// TwinCAT 3 PLC project SxrVacPlc
// ProgramVersion: 3.1.4022.4
// libraries:
//   L2SI Vacuum Library, * (SLAC)
//   LCLS General, * (SLAC)
//   Tc2_Standard, * (Beckhoff Automation GmbH)
//   Tc2_System, * (Beckhoff Automation GmbH)
//   Tc2_Utilities, * (Beckhoff Automation GmbH)
//   Tc3_Module, * (Beckhoff Automation GmbH)
// project tree:
//   GVLs/ GVL_SXR_VAC.TcGVL, GVL_Variables.TcGVL
//   / PlcTask.TcTTO
//   POUs/ MAIN.TcPOU, PRG_DIAGNOSTIC.TcPOU, PRG_SXR_VAC.TcPOU
// real-time tasks:
//   TASK PlcTask: cycle T#10ms, priority 20, ADS port 350
//   TASK SimTask: cycle T#10ms, priority 21, ADS port 351
// I/O:
//   DEVICE =+-EK1200_00_00-CPU/EtherCAT1, AmsNetId 10.0.1.49.2.1
//     =+-EK1200_00_00 [EK1200-5000 EtherCAT Power supply (2A E-Bus)]
//       =+-ES3064_00_01 [EL3064 4Ch. Ana. Input 0-10V]
//       =+-ES1004_00_02 [EL1004 4Ch. Dig. Input 24V, 3ms]
//       =+-EL2794_00_03 [EL2794 4Ch. Dig. Output 24V AC/DC, 2A, short-circuit-proof]
//       =+-ES3064_00_04 [EL3064 4Ch. Ana. Input 0-10V]
//       =+-ES1004_00_05 [EL1004 4Ch. Dig. Input 24V, 3ms]
//       =+-EL2794_00_06 [EL2794 4Ch. Dig. Output 24V AC/DC, 2A, short-circuit-proof]
//       =+-EL9410_00_07 [EL9410 E-Bus Power Supplier  (Diagnostics)]
//       =+-ES3064_00_08 [EL3064 4Ch. Ana. Input 0-10V]
//       =+-ES1004_00_09 [EL1004 4Ch. Dig. Input 24V, 3ms]
//       =+-EL2794_00_10 [EL2794 4Ch. Dig. Output 24V AC/DC, 2A, short-circuit-proof]
//       =+-ES3064_00_11 [EL3064 4Ch. Ana. Input 0-10V]
//       =+-ES1004_00_12 [EL1004 4Ch. Dig. Input 24V, 3ms]
//       =+-EL2794_00_13 [EL2794 4Ch. Dig. Output 24V AC/DC, 2A, short-circuit-proof]
//       =+-EK1110_00_14 [EK1110 EtherCAT extension]
//     =+-EK1100_01_00 [EK1100 EtherCAT Coupler (2A E-Bus)]
//       =+-ES3068_01_01 [EL3068 8Ch. Ana. Input 0-10V]
//       =+-EL2798_01_02 [EL2798 8Ch. Dig. Output 24V AC/DC, 2A, potential-free]
//       =+-ES9187_01_03 [EL9187 Potential Connection, 8 x Ground]
//       =+-ES3068_01_04 [EL3068 8Ch. Ana. Input 0-10V]
//       =+-ES3068_01_05 [EL3068 8Ch. Ana. Input 0-10V]
//       =+-EL2798_01_06 [EL2798 8Ch. Dig. Output 24V AC/DC, 2A, potential-free]
//       =+-ES9187_01_07 [EL9187 Potential Connection, 8 x Ground]
//       =+-ES3068_01_08 [EL3068 8Ch. Ana. Input 0-10V]
//       =+-EL9410_01_09 [EL9410 E-Bus Power Supplier  (Diagnostics)]
//       =+-EL2202_01_10 [EL2022 2Ch. Dig. Output 24V, 2A]
//       =+-EL6695_01_11 [EL6695 EtherCAT Bridge terminal (Primary)]
//       =+-EL6695_01_12 [EL6695 EtherCAT Bridge terminal (Primary)]
//       =+-EL6695_01_13 [EL6695 EtherCAT Bridge terminal (Primary)]
//       =+-EL6695_01_14 [EL6695 EtherCAT Bridge terminal (Primary)]
//     =+-EK1100_02_00 [EK1100 EtherCAT Coupler (2A E-Bus)]
//       =+-EL3064_02_01 [EL3064 4Ch. Ana. Input 0-10V]
//       =+-EL9070_02_02 [EL9070 Shield terminal]
//       =+-ES1008_02_03 [EL1008 8Ch. Dig. Input 24V, 3ms]
//       =+-ES9184_02_04 [EL9184 Potential Connection, 8 x 24V, 8 x Ground]
//       =+-ES2008_02_05 [EL2008 8Ch. Dig. Output 24V, 0.5A]
//       =+-EL2798_02_06 [EL2798 8Ch. Dig. Output 24V AC/DC, 2A, potential-free]
//     =+-EK1100_03_00 [EK1100 EtherCAT Coupler (2A E-Bus)]
//       =+-ES1004_03_01 [EL1004 4Ch. Dig. Input 24V, 3ms]
//       =+-ES2004_03_02 [EL2004 4Ch. Dig. Output 24V, 0.5A]
//       =+-ES2004_03_03 [EL2004 4Ch. Dig. Output 24V, 0.5A]
//       =+-ES1004_03_04 [EL1008 8Ch. Dig. Input 24V, 3ms]
//       =+-EL3064_03_05 [EL3064 4Ch. Ana. Input 0-10V]
//       =+-EL9070_03_06 [EL9070 Shield terminal]
//       =+-ES1008_03_07 [EL1008 8Ch. Dig. Input 24V, 3ms]
//       =+-ES9184_03_08 [EL9184 Potential Connection, 8 x 24V, 8 x Ground]
//       =+-ES2008_03_09 [EL2008 8Ch. Dig. Output 24V, 0.5A]
//       =+-EL2798_03_10 [EL2798 8Ch. Dig. Output 24V AC/DC, 2A, potential-free]
//     =+-EP2338_04_00 [EP2338-0002 8 Ch. Dig. Input/Output 24V, 0,5A, M12]
//     =+-EP2338_05_00 [EP2338-0002 8 Ch. Dig. Input/Output 24V, 0,5A, M12]
//     =+-EK1100_05_01 [EK1100 EtherCAT Coupler (2A E-Bus)]
//       =+-ES1004_05_02 [EL1004 4Ch. Dig. Input 24V, 3ms]
//       =+-ES2202_05_03 [EL2202 2Ch. Dig. Output 24V, 0.5A]
//       =+-ES2202_05_04 [EL2202 2Ch. Dig. Output 24V, 0.5A]
//       =+-ES9505_05_05 [EL9505 Power supply terminal 5V]
//       =+-ES1124_05_06 [EL1124 4Ch. Dig. Input 5V, 10µs, Sensor Power]
//     =+-EP2338_06_00 [EP2338-0002 8 Ch. Dig. Input/Output 24V, 0,5A, M12]
//     =+-EP2338_07_00 [EP2338-0002 8 Ch. Dig. Input/Output 24V, 0,5A, M12]
//     =+-EP3174_07_01 [EP3174-0002 4Ch. Ana. Input +/-10V, 0-10V, 0/4-20mA configurable]
//     =+-EP2624_07_02 [EP2624-0002 4Ch. Relay Output, NO (125V AC / 30V DC)]
//     =+-EP2338_08_00 [EP2338-0002 8 Ch. Dig. Input/Output 24V, 0,5A, M12]
//     =+-EP3174_08_01 [EP3174-0002 4Ch. Ana. Input +/-10V, 0-10V, 0/4-20mA configurable]
//     =+-EP2624_08_02 [EP2624-0002 4Ch. Relay Output, NO (125V AC / 30V DC)]
//     =+-EP3174_09_00 [EP3174-0002 4Ch. Ana. Input +/-10V, 0-10V, 0/4-20mA configurable]
//     =+-EP2624_09_01 [EP2624-0002 4Ch. Relay Output, NO (125V AC / 30V DC)]
//     =+-EP2338_09_02 [EP2338-0002 8 Ch. Dig. Input/Output 24V, 0,5A, M12]
//     =+-EP2338_09_03 [EP2338-0002 8 Ch. Dig. Input/Output 24V, 0,5A, M12]
//     =+-EP3174_10_00 [EP3174-0002 4Ch. Ana. Input +/-10V, 0-10V, 0/4-20mA configurable]
//     =+-EP2624_10_01 [EP2624-0002 4Ch. Relay Output, NO (125V AC / 30V DC)]
//     =+-EP2338_10_02 [EP2338-0002 8 Ch. Dig. Input/Output 24V, 0,5A, M12]
//     =+-EP3174_11_00 [EP3174-0002 4Ch. Ana. Input +/-10V, 0-10V, 0/4-20mA configurable]
//     =+-EP2624_11_01 [EP2624-0002 4Ch. Relay Output, NO (125V AC / 30V DC)]
//     =+-EP2338_11_02 [EP2338-0002 8 Ch. Dig. Input/Output 24V, 0,5A, M12]
//     =+-EK1100_11_03 [EK1100 EtherCAT Coupler (2A E-Bus)]
//       =+-ES1004_11_04 [EL1004 4Ch. Dig. Input 24V, 3ms]
//       =+-ES2202_11_05 [EL2202 2Ch. Dig. Output 24V, 0.5A]
//       =+-ES2202_11_06 [EL2202 2Ch. Dig. Output 24V, 0.5A]
//       =+-ES9505_11_07 [EL9505 Power supply terminal 5V]
//       =+-ES1124_11_08 [EL1124 4Ch. Dig. Input 5V, 10µs, Sensor Power]
//     =+-EP3174_12_00 [EP3174-0002 4Ch. Ana. Input +/-10V, 0-10V, 0/4-20mA configurable]
//     =+-EP2624_12_01 [EP2624-0002 4Ch. Relay Output, NO (125V AC / 30V DC)]
//     =+-EP3174_13_00 [EP3174-0002 4Ch. Ana. Input +/-10V, 0-10V, 0/4-20mA configurable]
//     =+-EP2624_13_01 [EP2624-0002 4Ch. Relay Output, NO (125V AC / 30V DC)]
//     =+-EP2338_14_00 [EP2338-0002 8 Ch. Dig. Input/Output 24V, 0,5A, M12]
//     =+-EP3174_14_01 [EP3174-0002 4Ch. Ana. Input +/-10V, 0-10V, 0/4-20mA configurable]
//     =+-EP2624_14_02 [EP2624-0002 4Ch. Relay Output, NO (125V AC / 30V DC)]
//     =+-EK1100_15_00 [EK1100 EtherCAT Coupler (2A E-Bus)]
//       =+-ES3064_15_01 [EL3064 4Ch. Ana. Input 0-10V]
//       =+-ES1004_15_02 [EL1004 4Ch. Dig. Input 24V, 3ms]
//       =+-EL2794_15_03 [EL2794 4Ch. Dig. Output 24V AC/DC, 2A, short-circuit-proof]
//       =+-ES3064_15_04 [EL3064 4Ch. Ana. Input 0-10V]
//       =+-ES1004_15_05 [EL1004 4Ch. Dig. Input 24V, 3ms]
//       =+-EL2794_15_06 [EL2794 4Ch. Dig. Output 24V AC/DC, 2A, short-circuit-proof]
//   DEVICE SimDevice 2 (EtherCAT Simulation), AmsNetId 10.0.1.49.3.1
//     =+-ES3064_00_01 // EL3064-0000-0020
//     =+-ES1004_00_02 // EL1004-0000-0019
//     =+-EL2794_00_03 // EL2794-0000-0016
//     =+-ES3064_00_04 // EL3064-0000-0020
//     =+-ES1004_00_05 // EL1004-0000-0019
//     =+-EL2794_00_06 // EL2794-0000-0016
//     =+-EL9410_00_07 // EL9410-0000-0017
//     =+-ES3064_00_08 // EL3064-0000-0020
//     =+-ES1004_00_09 // EL1004-0000-0019
//     =+-EL2794_00_10 // EL2794-0000-0016
//     =+-ES3064_00_11 // EL3064-0000-0020
//     =+-ES1004_00_12 // EL1004-0000-0019
//     =+-EL2794_00_13 // EL2794-0000-0016
//     =+-EK1110_00_14 // EK1110-0000-0017
//     =+-EK1100_01_00 // EK1100-0000-0018
//     =+-ES3068_01_01 // EL3068-0000-0020
//     =+-EL2798_01_02 // EL2798-0000-0018
//     =+-ES3068_01_04 // EL3068-0000-0020
//     =+-ES3068_01_05 // EL3068-0000-0020
//     =+-EL2798_01_06 // EL2798-0000-0018
//     =+-ES3068_01_08 // EL3068-0000-0020
//     =+-EL9410_01_09 // EL9410-0000-0017
//     =+-EL2202_01_10 // EL2022-0000-0018
//     =+-EL6695_01_11 // EL6695-0000-0005
//     =+-EL6695_01_12 // EL6695-0000-0005
//     =+-EL6695_01_13 // EL6695-0000-0005
//     =+-EL6695_01_14 // EL6695-0000-0005
//     =+-EK1100_02_00 // EK1100-0000-0018
//     =+-EL3064_02_01 // EL3064-0000-0020
//     =+-ES1008_02_03 // EL1008-0000-0018
//     =+-ES2008_02_05 // EL2008-0000-0018
//     =+-EL2798_02_06 // EL2798-0000-0018
//     =+-EK1100_03_00 // EK1100-0000-0018
//     =+-ES1004_03_01 // EL1004-0000-0019
//     =+-ES2004_03_02 // EL2004-0000-0018
//     =+-ES2004_03_03 // EL2004-0000-0018
//     =+-ES1004_03_04 // EL1008-0000-0018
//     =+-EL3064_03_05 // EL3064-0000-0020
//     =+-ES1008_03_07 // EL1008-0000-0018
//     =+-ES2008_03_09 // EL2008-0000-0018
//     =+-EL2798_03_10 // EL2798-0000-0018
//     =+-EP2338_04_00 // EP2338-0002-0023
//     =+-EP2338_05_00 // EP2338-0002-0023
//     =+-EK1100_05_01 // EK1100-0000-0018
//     =+-ES1004_05_02 // EL1004-0000-0019
//     =+-ES2202_05_03 // EL2202-0000-0019
//     =+-ES2202_05_04 // EL2202-0000-0019
//     =+-ES9505_05_05 // EL9505-0000-0018
//     =+-ES1124_05_06 // EL1124-0000-0018
//     =+-EP2338_06_00 // EP2338-0002-0023
//     =+-EP2338_07_00 // EP2338-0002-0023
//     =+-EP3174_07_01 // EP3174-0002-0023
//     =+-EP2624_07_02 // EP2624-0002-0019
//     =+-EP2338_08_00 // EP2338-0002-0023
//     =+-EP3174_08_01 // EP3174-0002-0023
//     =+-EP2624_08_02 // EP2624-0002-0019
//     =+-EP3174_09_00 // EP3174-0002-0023
//     =+-EP2624_09_01 // EP2624-0002-0019
//     =+-EP2338_09_02 // EP2338-0002-0023
//     =+-EP2338_09_03 // EP2338-0002-0023
//     =+-EP3174_10_00 // EP3174-0002-0023
//     =+-EP2624_10_01 // EP2624-0002-0019
//     =+-EP2338_10_02 // EP2338-0002-0023
//     =+-EP3174_11_00 // EP3174-0002-0023
//     =+-EP2624_11_01 // EP2624-0002-0019
//     =+-EP2338_11_02 // EP2338-0002-0023
//     =+-EK1100_11_03 // EK1100-0000-0018
//     =+-ES1004_11_04 // EL1004-0000-0019
//     =+-ES2202_11_05 // EL2202-0000-0019
//     =+-ES2202_11_06 // EL2202-0000-0019
//     =+-ES9505_11_07 // EL9505-0000-0018
//     =+-ES1124_11_08 // EL1124-0000-0018
//     =+-EP3174_12_00 // EP3174-0002-0023
//     =+-EP2624_12_01 // EP2624-0002-0019
//     =+-EP3174_13_00 // EP3174-0002-0023
//     =+-EP2624_13_01 // EP2624-0002-0019
//     =+-EP2338_14_00 // EP2338-0002-0023
//     =+-EP3174_14_01 // EP3174-0002-0023
//     =+-EP2624_14_02 // EP2624-0002-0019
//     =+-EK1100_15_00 // EK1100-0000-0018
//     =+-ES3064_15_01 // EL3064-0000-0020
//     =+-ES1004_15_02 // EL1004-0000-0019
//     =+-EL2794_15_03 // EL2794-0000-0016
//     =+-ES3064_15_04 // EL3064-0000-0020
//     =+-ES1004_15_05 // EL1004-0000-0019
//     =+-EL2794_15_06 // EL2794-0000-0016
// variable links:
//   SxrVacPlc/SxrVacPlc Instance <-> =+-EK1200_00_00-CPU/EtherCAT1/=+-EK1100_01_00/=+-EL2798_01_02
//     PlcTask Outputs/GVL_SXR_VAC.fb_DMPS_GCC_1.q_xHV_DIS <-> Channel 1/GVL_SXR_VAC.fb_DMPS_GCC_1.q_xHV_DIS
//     PlcTask Outputs/GVL_SXR_VAC.fb_IM2K0_XTES_GCC_1.q_xHV_DIS <-> Channel 2/GVL_SXR_VAC.fb_IM2K0_XTES_GCC_1.q_xHV_DIS
//     PlcTask Outputs/GVL_SXR_VAC.fb_PCPM3B_GFS_1.q_xHV_DIS <-> Channel 5/GVL_SXR_VAC.fb_PCPM3B_GFS_1.q_xHV_DIS
//     PlcTask Outputs/GVL_SXR_VAC.fb_SL1K0_GCC_1.q_xHV_DIS <-> Channel 4/GVL_SXR_VAC.fb_SL1K0_GCC_1.q_xHV_DIS
//   SxrVacPlc/SxrVacPlc Instance <-> =+-EK1200_00_00-CPU/EtherCAT1/=+-EK1100_01_00/=+-EL2798_01_06
//     PlcTask Outputs/GVL_SXR_VAC.fb_MR1K1_BEND_GCC_1.q_xHV_DIS <-> Channel 5/GVL_SXR_VAC.fb_MR1K1_BEND_GCC_1.q_xHV_DIS
//     PlcTask Outputs/GVL_SXR_VAC.fb_PA1K0_GCC_1.q_xHV_DIS <-> Channel 4/GVL_SXR_VAC.fb_PA1K0_GCC_1.q_xHV_DIS
//     PlcTask Outputs/GVL_SXR_VAC.fb_TV2K0_GCC_1.q_xHV_DIS <-> Channel 1/GVL_SXR_VAC.fb_TV2K0_GCC_1.q_xHV_DIS
//     PlcTask Outputs/GVL_SXR_VAC.fb_TV2K0_GCC_2.q_xHV_DIS <-> Channel 2/GVL_SXR_VAC.fb_TV2K0_GCC_2.q_xHV_DIS
//   SxrVacPlc/SxrVacPlc Instance <-> =+-EK1200_00_00-CPU/EtherCAT1/=+-EK1100_01_00/=+-ES3068_01_01
//     PlcTask Inputs/GVL_SXR_VAC.fb_DMPS_GCC_1.i_iPRESS_R <-> AI Standard Channel 1/GVL_SXR_VAC.fb_DMPS_GCC_1.i_iPRESS_R
//     PlcTask Inputs/GVL_SXR_VAC.fb_DMPS_GPI_1.i_iPRESS_R <-> AI Standard Channel 5/GVL_SXR_VAC.fb_DMPS_GPI_1.i_iPRESS_R
//     PlcTask Inputs/GVL_SXR_VAC.fb_IM2K0_XTES_GCC_1.i_iPRESS_R <-> AI Standard Channel 3/GVL_SXR_VAC.fb_IM2K0_XTES_GCC_1.i_iPRESS_R
//     PlcTask Inputs/GVL_SXR_VAC.fb_IM2K0_XTES_GPI_1.i_iPRESS_R <-> AI Standard Channel 6/GVL_SXR_VAC.fb_IM2K0_XTES_GPI_1.i_iPRESS_R
//   SxrVacPlc/SxrVacPlc Instance <-> =+-EK1200_00_00-CPU/EtherCAT1/=+-EK1100_01_00/=+-ES3068_01_04
//     PlcTask Inputs/GVL_SXR_VAC.fb_PCPM3B_GFS_1.i_iPRESS_R <-> AI Standard Channel 3/GVL_SXR_VAC.fb_PCPM3B_GFS_1.i_iPRESS_R
//     PlcTask Inputs/GVL_SXR_VAC.fb_SL1K0_GCC_1.i_iPRESS_R <-> AI Standard Channel 1/GVL_SXR_VAC.fb_SL1K0_GCC_1.i_iPRESS_R
//     PlcTask Inputs/GVL_SXR_VAC.fb_SL1K0_GPI_1.i_iPRESS_R <-> AI Standard Channel 5/GVL_SXR_VAC.fb_SL1K0_GPI_1.i_iPRESS_R
//   SxrVacPlc/SxrVacPlc Instance <-> =+-EK1200_00_00-CPU/EtherCAT1/=+-EK1100_01_00/=+-ES3068_01_05
//     PlcTask Inputs/GVL_SXR_VAC.fb_TV2K0_GCC_1.i_iPRESS_R <-> AI Standard Channel 1/GVL_SXR_VAC.fb_TV2K0_GCC_1.i_iPRESS_R
//     PlcTask Inputs/GVL_SXR_VAC.fb_TV2K0_GCC_2.i_iPRESS_R <-> AI Standard Channel 3/GVL_SXR_VAC.fb_TV2K0_GCC_2.i_iPRESS_R
//     PlcTask Inputs/GVL_SXR_VAC.fb_TV2K0_GPI_1.i_iPRESS_R <-> AI Standard Channel 5/GVL_SXR_VAC.fb_TV2K0_GPI_1.i_iPRESS_R
//     PlcTask Inputs/GVL_SXR_VAC.fb_TV2K0_GPI_2.i_iPRESS_R <-> AI Standard Channel 6/GVL_SXR_VAC.fb_TV2K0_GPI_2.i_iPRESS_R
//   SxrVacPlc/SxrVacPlc Instance <-> =+-EK1200_00_00-CPU/EtherCAT1/=+-EK1100_01_00/=+-ES3068_01_08
//     PlcTask Inputs/GVL_SXR_VAC.fb_MR1K1_BEND_GCC_1.i_iPRESS_R <-> AI Standard Channel 3/GVL_SXR_VAC.fb_MR1K1_BEND_GCC_1.i_iPRESS_R
//     PlcTask Inputs/GVL_SXR_VAC.fb_MR1K1_BEND_GPI_1.i_iPRESS_R <-> AI Standard Channel 6/GVL_SXR_VAC.fb_MR1K1_BEND_GPI_1.i_iPRESS_R
//     PlcTask Inputs/GVL_SXR_VAC.fb_PA1K0_GCC_1.i_iPRESS_R <-> AI Standard Channel 1/GVL_SXR_VAC.fb_PA1K0_GCC_1.i_iPRESS_R
//     PlcTask Inputs/GVL_SXR_VAC.fb_PA1K0_GPI_1.i_iPRESS_R <-> AI Standard Channel 5/GVL_SXR_VAC.fb_PA1K0_GPI_1.i_iPRESS_R
//   SxrVacPlc/SxrVacPlc Instance <-> =+-EK1200_00_00-CPU/EtherCAT1/=+-EK1100_03_00/=+-ES1004_03_01
//     PlcTask Inputs/GVL_SXR_VAC.fb_EM1K0_GMD_VGC_1.i_xClsLS <-> Channel 4/GVL_SXR_VAC.fb_EM1K0_GMD_VGC_1.i_xClsLS
//     PlcTask Inputs/GVL_SXR_VAC.fb_EM1K0_GMD_VGC_1.i_xOpnLS <-> Channel 3/GVL_SXR_VAC.fb_EM1K0_GMD_VGC_1.i_xOpnLS
//     PlcTask Inputs/GVL_SXR_VAC.fb_RTDSK0_VGC_1.i_xClsLS <-> Channel 2/GVL_SXR_VAC.fb_RTDSK0_VGC_1.i_xClsLS
//     PlcTask Inputs/GVL_SXR_VAC.fb_RTDSK0_VGC_1.i_xOpnLS <-> Channel 1/GVL_SXR_VAC.fb_RTDSK0_VGC_1.i_xOpnLS
//   SxrVacPlc/SxrVacPlc Instance <-> =+-EK1200_00_00-CPU/EtherCAT1/=+-EK1100_03_00/=+-ES1004_03_04
//     PlcTask Inputs/GVL_SXR_VAC.fb_AT1K0_GAS_VGC_1.i_xClsLS <-> Channel 2/GVL_SXR_VAC.fb_AT1K0_GAS_VGC_1.i_xClsLS
//     PlcTask Inputs/GVL_SXR_VAC.fb_AT1K0_GAS_VGC_1.i_xOpnLS <-> Channel 1/GVL_SXR_VAC.fb_AT1K0_GAS_VGC_1.i_xOpnLS
//   SxrVacPlc/SxrVacPlc Instance <-> =+-EK1200_00_00-CPU/EtherCAT1/=+-EK1100_03_00/=+-ES2004_03_02
//     PlcTask Outputs/GVL_SXR_VAC.fb_EM1K0_GMD_VGC_1.q_xOPN_DO <-> Channel 3/GVL_SXR_VAC.fb_EM1K0_GMD_VGC_1.q_xOPN_DO
//     PlcTask Outputs/GVL_SXR_VAC.fb_RTDSK0_VGC_1.q_xOPN_DO <-> Channel 1/GVL_SXR_VAC.fb_RTDSK0_VGC_1.q_xOPN_DO
//   SxrVacPlc/SxrVacPlc Instance <-> =+-EK1200_00_00-CPU/EtherCAT1/=+-EK1100_03_00/=+-ES2004_03_03
//     PlcTask Outputs/GVL_SXR_VAC.fb_AT1K0_GAS_VGC_1.q_xOPN_DO <-> Channel 1/GVL_SXR_VAC.fb_AT1K0_GAS_VGC_1.q_xOPN_DO
//   SxrVacPlc/SxrVacPlc Instance <-> =+-EK1200_00_00-CPU/EtherCAT1/=+-EK1100_15_00/=+-EL2794_15_03
//     PlcTask Outputs/GVL_SXR_VAC.fb_MR1K4_SOMS_PIP_1.q_xHVEna_DO <-> Channel 1/GVL_SXR_VAC.fb_MR1K4_SOMS_PIP_1.q_xHVEna_DO
//     PlcTask Outputs/GVL_SXR_VAC.fb_ST1K4_TEST_PIP_1.q_xHVEna_DO <-> Channel 2/GVL_SXR_VAC.fb_ST1K4_TEST_PIP_1.q_xHVEna_DO
//     PlcTask Outputs/GVL_SXR_VAC.fb_ST2K4_BCS_PIP_1.q_xHVEna_DO <-> Channel 3/GVL_SXR_VAC.fb_ST2K4_BCS_PIP_1.q_xHVEna_DO
//     PlcTask Outputs/GVL_SXR_VAC.fb_ST3K4_PPS_PIP_1.q_xHVEna_DO <-> Channel 4/GVL_SXR_VAC.fb_ST3K4_PPS_PIP_1.q_xHVEna_DO
//   SxrVacPlc/SxrVacPlc Instance <-> =+-EK1200_00_00-CPU/EtherCAT1/=+-EK1100_15_00/=+-EL2794_15_06
//     PlcTask Outputs/GVL_SXR_VAC.fb_PC4K4_XTES_PIP_1.q_xHVEna_DO <-> Channel 1/GVL_SXR_VAC.fb_PC4K4_XTES_PIP_1.q_xHVEna_DO
//   SxrVacPlc/SxrVacPlc Instance <-> =+-EK1200_00_00-CPU/EtherCAT1/=+-EK1100_15_00/=+-ES1004_15_02
//     PlcTask Inputs/GVL_SXR_VAC.fb_MR1K4_SOMS_PIP_1.i_xSP_DI <-> Channel 1/GVL_SXR_VAC.fb_MR1K4_SOMS_PIP_1.i_xSP_DI
//     PlcTask Inputs/GVL_SXR_VAC.fb_ST1K4_TEST_PIP_1.i_xSP_DI <-> Channel 2/GVL_SXR_VAC.fb_ST1K4_TEST_PIP_1.i_xSP_DI
//     PlcTask Inputs/GVL_SXR_VAC.fb_ST2K4_BCS_PIP_1.i_xSP_DI <-> Channel 3/GVL_SXR_VAC.fb_ST2K4_BCS_PIP_1.i_xSP_DI
//     PlcTask Inputs/GVL_SXR_VAC.fb_ST3K4_PPS_PIP_1.i_xSP_DI <-> Channel 4/GVL_SXR_VAC.fb_ST3K4_PPS_PIP_1.i_xSP_DI
//   SxrVacPlc/SxrVacPlc Instance <-> =+-EK1200_00_00-CPU/EtherCAT1/=+-EK1100_15_00/=+-ES1004_15_05
//     PlcTask Inputs/GVL_SXR_VAC.fb_PC4K4_XTES_PIP_1.i_xSP_DI <-> Channel 1/GVL_SXR_VAC.fb_PC4K4_XTES_PIP_1.i_xSP_DI
//   SxrVacPlc/SxrVacPlc Instance <-> =+-EK1200_00_00-CPU/EtherCAT1/=+-EK1100_15_00/=+-ES3064_15_01
//     PlcTask Inputs/GVL_SXR_VAC.fb_MR1K4_SOMS_PIP_1.i_iPRESS <-> AI Standard Channel 1/GVL_SXR_VAC.fb_MR1K4_SOMS_PIP_1.i_iPRESS
//     PlcTask Inputs/GVL_SXR_VAC.fb_ST1K4_TEST_PIP_1.i_iPRESS <-> AI Standard Channel 2/GVL_SXR_VAC.fb_ST1K4_TEST_PIP_1.i_iPRESS
//     PlcTask Inputs/GVL_SXR_VAC.fb_ST2K4_BCS_PIP_1.i_iPRESS <-> AI Standard Channel 3/GVL_SXR_VAC.fb_ST2K4_BCS_PIP_1.i_iPRESS
//     PlcTask Inputs/GVL_SXR_VAC.fb_ST3K4_PPS_PIP_1.i_iPRESS <-> AI Standard Channel 4/GVL_SXR_VAC.fb_ST3K4_PPS_PIP_1.i_iPRESS
//   SxrVacPlc/SxrVacPlc Instance <-> =+-EK1200_00_00-CPU/EtherCAT1/=+-EK1100_15_00/=+-ES3064_15_04
//     PlcTask Inputs/GVL_SXR_VAC.fb_PC4K4_XTES_PIP_1.i_iPRESS <-> AI Standard Channel 1/GVL_SXR_VAC.fb_PC4K4_XTES_PIP_1.i_iPRESS
//   SxrVacPlc/SxrVacPlc Instance <-> =+-EK1200_00_00-CPU/EtherCAT1/=+-EK1200_00_00/=+-EL2794_00_03
//     PlcTask Outputs/GVL_SXR_VAC.fb_RTDSK0_PIP_{1..4}.q_xHVEna_DO <-> Channel {1..4}/GVL_SXR_VAC.fb_RTDSK0_PIP_{1..4}.q_xHVEna_DO  (4 links)
//   SxrVacPlc/SxrVacPlc Instance <-> =+-EK1200_00_00-CPU/EtherCAT1/=+-EK1200_00_00/=+-EL2794_00_06
//     PlcTask Outputs/GVL_SXR_VAC.fb_PCPM3B_PIP_1.q_xHVEna_DO <-> Channel 2/GVL_SXR_VAC.fb_PCPM3B_PIP_1.q_xHVEna_DO
//     PlcTask Outputs/GVL_SXR_VAC.fb_RTDSK0_PIP_5.q_xHVEna_DO <-> Channel 1/GVL_SXR_VAC.fb_RTDSK0_PIP_5.q_xHVEna_DO
//   SxrVacPlc/SxrVacPlc Instance <-> =+-EK1200_00_00-CPU/EtherCAT1/=+-EK1200_00_00/=+-EL2794_00_10
//     PlcTask Outputs/GVL_SXR_VAC.fb_MR1K1_BEND_PIP_1.q_xHVEna_DO <-> Channel 3/GVL_SXR_VAC.fb_MR1K1_BEND_PIP_1.q_xHVEna_DO
//     PlcTask Outputs/GVL_SXR_VAC.fb_MR1K3_TXI_PIP_1.q_xHVEna_DO <-> Channel 4/GVL_SXR_VAC.fb_MR1K3_TXI_PIP_1.q_xHVEna_DO
//     PlcTask Outputs/GVL_SXR_VAC.fb_PA1K0_PIP_1.q_xHVEna_DO <-> Channel 1/GVL_SXR_VAC.fb_PA1K0_PIP_1.q_xHVEna_DO
//   SxrVacPlc/SxrVacPlc Instance <-> =+-EK1200_00_00-CPU/EtherCAT1/=+-EK1200_00_00/=+-EL2794_00_13
//     PlcTask Outputs/GVL_SXR_VAC.fb_MR2K3_TXI_PIP_1.q_xHVEna_DO <-> Channel 1/GVL_SXR_VAC.fb_MR2K3_TXI_PIP_1.q_xHVEna_DO
//     PlcTask Outputs/GVL_SXR_VAC.fb_SP1K1_MONO_PIP_1.q_xHVEna_DO <-> Channel 2/GVL_SXR_VAC.fb_SP1K1_MONO_PIP_1.q_xHVEna_DO
//     PlcTask Outputs/GVL_SXR_VAC.fb_SP1K1_MONO_PIP_2.q_xHVEna_DO <-> Channel 3/GVL_SXR_VAC.fb_SP1K1_MONO_PIP_2.q_xHVEna_DO
//     PlcTask Outputs/GVL_SXR_VAC.fb_TV3K0_PIP_1.q_xHVEna_DO <-> Channel 4/GVL_SXR_VAC.fb_TV3K0_PIP_1.q_xHVEna_DO
//   SxrVacPlc/SxrVacPlc Instance <-> =+-EK1200_00_00-CPU/EtherCAT1/=+-EK1200_00_00/=+-ES1004_00_02
//     PlcTask Inputs/GVL_SXR_VAC.fb_RTDSK0_PIP_{1..4}.i_xSP_DI <-> Channel {1..4}/GVL_SXR_VAC.fb_RTDSK0_PIP_{1..4}.i_xSP_DI  (4 links)
//   SxrVacPlc/SxrVacPlc Instance <-> =+-EK1200_00_00-CPU/EtherCAT1/=+-EK1200_00_00/=+-ES1004_00_05
//     PlcTask Inputs/GVL_SXR_VAC.fb_PCPM3B_PIP_1.i_xSP_DI <-> Channel 2/GVL_SXR_VAC.fb_PCPM3B_PIP_1.i_xSP_DI
//     PlcTask Inputs/GVL_SXR_VAC.fb_RTDSK0_PIP_5.i_xSP_DI <-> Channel 1/GVL_SXR_VAC.fb_RTDSK0_PIP_5.i_xSP_DI
//   SxrVacPlc/SxrVacPlc Instance <-> =+-EK1200_00_00-CPU/EtherCAT1/=+-EK1200_00_00/=+-ES1004_00_09
//     PlcTask Inputs/GVL_SXR_VAC.fb_MR1K1_BEND_PIP_1.i_xSP_DI <-> Channel 3/GVL_SXR_VAC.fb_MR1K1_BEND_PIP_1.i_xSP_DI
//     PlcTask Inputs/GVL_SXR_VAC.fb_MR1K3_TXI_PIP_1.i_xSP_DI <-> Channel 4/GVL_SXR_VAC.fb_MR1K3_TXI_PIP_1.i_xSP_DI
//     PlcTask Inputs/GVL_SXR_VAC.fb_PA1K0_PIP_1.i_xSP_DI <-> Channel 1/GVL_SXR_VAC.fb_PA1K0_PIP_1.i_xSP_DI
//   SxrVacPlc/SxrVacPlc Instance <-> =+-EK1200_00_00-CPU/EtherCAT1/=+-EK1200_00_00/=+-ES1004_00_12
//     PlcTask Inputs/GVL_SXR_VAC.fb_MR2K3_TXI_PIP_1.i_xSP_DI <-> Channel 1/GVL_SXR_VAC.fb_MR2K3_TXI_PIP_1.i_xSP_DI
//     PlcTask Inputs/GVL_SXR_VAC.fb_SP1K1_MONO_PIP_1.i_xSP_DI <-> Channel 2/GVL_SXR_VAC.fb_SP1K1_MONO_PIP_1.i_xSP_DI
//     PlcTask Inputs/GVL_SXR_VAC.fb_SP1K1_MONO_PIP_2.i_xSP_DI <-> Channel 3/GVL_SXR_VAC.fb_SP1K1_MONO_PIP_2.i_xSP_DI
//     PlcTask Inputs/GVL_SXR_VAC.fb_TV3K0_PIP_1.i_xSP_DI <-> Channel 4/GVL_SXR_VAC.fb_TV3K0_PIP_1.i_xSP_DI
//   SxrVacPlc/SxrVacPlc Instance <-> =+-EK1200_00_00-CPU/EtherCAT1/=+-EK1200_00_00/=+-ES3064_00_01
//     PlcTask Inputs/GVL_SXR_VAC.fb_RTDSK0_PIP_{1..4}.i_iPRESS <-> AI Standard Channel {1..4}/GVL_SXR_VAC.fb_RTDSK0_PIP_{1..4}.i_iPRESS  (4 links)
//   SxrVacPlc/SxrVacPlc Instance <-> =+-EK1200_00_00-CPU/EtherCAT1/=+-EK1200_00_00/=+-ES3064_00_04
//     PlcTask Inputs/GVL_SXR_VAC.fb_PCPM3B_PIP_1.i_iPRESS <-> AI Standard Channel 2/GVL_SXR_VAC.fb_PCPM3B_PIP_1.i_iPRESS
//     PlcTask Inputs/GVL_SXR_VAC.fb_RTDSK0_PIP_5.i_iPRESS <-> AI Standard Channel 1/GVL_SXR_VAC.fb_RTDSK0_PIP_5.i_iPRESS
//   SxrVacPlc/SxrVacPlc Instance <-> =+-EK1200_00_00-CPU/EtherCAT1/=+-EK1200_00_00/=+-ES3064_00_08
//     PlcTask Inputs/GVL_SXR_VAC.fb_MR1K1_BEND_PIP_1.i_iPRESS <-> AI Standard Channel 3/GVL_SXR_VAC.fb_MR1K1_BEND_PIP_1.i_iPRESS
//     PlcTask Inputs/GVL_SXR_VAC.fb_MR1K3_TXI_PIP_1.i_iPRESS <-> AI Standard Channel 4/GVL_SXR_VAC.fb_MR1K3_TXI_PIP_1.i_iPRESS
//     PlcTask Inputs/GVL_SXR_VAC.fb_PA1K0_PIP_1.i_iPRESS <-> AI Standard Channel 1/GVL_SXR_VAC.fb_PA1K0_PIP_1.i_iPRESS
//   SxrVacPlc/SxrVacPlc Instance <-> =+-EK1200_00_00-CPU/EtherCAT1/=+-EK1200_00_00/=+-ES3064_00_11
//     PlcTask Inputs/GVL_SXR_VAC.fb_MR2K3_TXI_PIP_1.i_iPRESS <-> AI Standard Channel 1/GVL_SXR_VAC.fb_MR2K3_TXI_PIP_1.i_iPRESS
//     PlcTask Inputs/GVL_SXR_VAC.fb_SP1K1_MONO_PIP_1.i_iPRESS <-> AI Standard Channel 2/GVL_SXR_VAC.fb_SP1K1_MONO_PIP_1.i_iPRESS
//     PlcTask Inputs/GVL_SXR_VAC.fb_SP1K1_MONO_PIP_2.i_iPRESS <-> AI Standard Channel 3/GVL_SXR_VAC.fb_SP1K1_MONO_PIP_2.i_iPRESS
//     PlcTask Inputs/GVL_SXR_VAC.fb_TV3K0_PIP_1.i_iPRESS <-> AI Standard Channel 4/GVL_SXR_VAC.fb_TV3K0_PIP_1.i_iPRESS
//   SxrVacPlc/SxrVacPlc Instance <-> =+-EK1200_00_00-CPU/EtherCAT1/=+-EP2338_04_00
//     PlcTask Inputs/GVL_SXR_VAC.fb_EM1K0_XGMD_VGC_1.i_xClsLS <-> Channel 2/GVL_SXR_VAC.fb_EM1K0_XGMD_VGC_1.i_xClsLS
//     PlcTask Inputs/GVL_SXR_VAC.fb_EM1K0_XGMD_VGC_2.i_xClsLS <-> Channel 6/GVL_SXR_VAC.fb_EM1K0_XGMD_VGC_2.i_xClsLS
//     PlcTask Inputs/GVL_SXR_VAC.fb_EM1K0_XGMD_VGC_1.i_xOpnLS <-> Channel 1/GVL_SXR_VAC.fb_EM1K0_XGMD_VGC_1.i_xOpnLS
//     PlcTask Inputs/GVL_SXR_VAC.fb_EM1K0_XGMD_VGC_2.i_xOpnLS <-> Channel 5/GVL_SXR_VAC.fb_EM1K0_XGMD_VGC_2.i_xOpnLS
//     PlcTask Outputs/GVL_SXR_VAC.fb_EM1K0_XGMD_VGC_1.q_xOPN_DO <-> Channel 11/GVL_SXR_VAC.fb_EM1K0_XGMD_VGC_1.q_xOPN_DO
//     PlcTask Outputs/GVL_SXR_VAC.fb_EM1K0_XGMD_VGC_2.q_xOPN_DO <-> Channel 15/GVL_SXR_VAC.fb_EM1K0_XGMD_VGC_2.q_xOPN_DO
//   SxrVacPlc/SxrVacPlc Instance <-> =+-EK1200_00_00-CPU/EtherCAT1/=+-EP2338_05_00
//     PlcTask Inputs/GVL_SXR_VAC.fb_TV2K0_VGC_1.i_xClsLS <-> Channel 2/GVL_SXR_VAC.fb_TV2K0_VGC_1.i_xClsLS
//     PlcTask Inputs/GVL_SXR_VAC.fb_TV2K0_VGC_1.i_xOpnLS <-> Channel 1/GVL_SXR_VAC.fb_TV2K0_VGC_1.i_xOpnLS
//     PlcTask Outputs/GVL_SXR_VAC.fb_TV2K0_VGC_1.q_xOPN_DO <-> Channel 11/GVL_SXR_VAC.fb_TV2K0_VGC_1.q_xOPN_DO
//   SxrVacPlc/SxrVacPlc Instance <-> =+-EK1200_00_00-CPU/EtherCAT1/=+-EP2338_06_00
//     PlcTask Inputs/GVL_SXR_VAC.fb_MR1K1_BEND_VGC_1.i_xClsLS <-> Channel 2/GVL_SXR_VAC.fb_MR1K1_BEND_VGC_1.i_xClsLS
//     PlcTask Inputs/GVL_SXR_VAC.fb_MR1K1_BEND_VGC_1.i_xOpnLS <-> Channel 1/GVL_SXR_VAC.fb_MR1K1_BEND_VGC_1.i_xOpnLS
//     PlcTask Outputs/GVL_SXR_VAC.fb_MR1K1_BEND_VGC_1.q_xOPN_DO <-> Channel 11/GVL_SXR_VAC.fb_MR1K1_BEND_VGC_1.q_xOPN_DO
//   SxrVacPlc/SxrVacPlc Instance <-> =+-EK1200_00_00-CPU/EtherCAT1/=+-EP2338_07_00
//     PlcTask Inputs/GVL_SXR_VAC.fb_MR1K3_TXI_VGC_1.i_xClsLS <-> Channel 2/GVL_SXR_VAC.fb_MR1K3_TXI_VGC_1.i_xClsLS
//     PlcTask Inputs/GVL_SXR_VAC.fb_MR1K3_TXI_VGC_1.i_xOpnLS <-> Channel 1/GVL_SXR_VAC.fb_MR1K3_TXI_VGC_1.i_xOpnLS
//     PlcTask Outputs/GVL_SXR_VAC.fb_MR1K3_TXI_VGC_1.q_xOPN_DO <-> Channel 11/GVL_SXR_VAC.fb_MR1K3_TXI_VGC_1.q_xOPN_DO
//   SxrVacPlc/SxrVacPlc Instance <-> =+-EK1200_00_00-CPU/EtherCAT1/=+-EP2338_08_00
//     PlcTask Inputs/GVL_SXR_VAC.fb_SP1K1_MONO_VGC_1.i_xClsLS <-> Channel 2/GVL_SXR_VAC.fb_SP1K1_MONO_VGC_1.i_xClsLS
//     PlcTask Inputs/GVL_SXR_VAC.fb_SP1K1_MONO_VGC_1.i_xOpnLS <-> Channel 1/GVL_SXR_VAC.fb_SP1K1_MONO_VGC_1.i_xOpnLS
//     PlcTask Outputs/GVL_SXR_VAC.fb_SP1K1_MONO_VGC_1.q_xOPN_DO <-> Channel 11/GVL_SXR_VAC.fb_SP1K1_MONO_VGC_1.q_xOPN_DO
//   SxrVacPlc/SxrVacPlc Instance <-> =+-EK1200_00_00-CPU/EtherCAT1/=+-EP2338_09_02
//     PlcTask Inputs/GVL_SXR_VAC.fb_SP1K1_MONO_VGC_2.i_xClsLS <-> Channel 2/GVL_SXR_VAC.fb_SP1K1_MONO_VGC_2.i_xClsLS
//     PlcTask Inputs/GVL_SXR_VAC.fb_SP1K1_MONO_VGC_2.i_xOpnLS <-> Channel 1/GVL_SXR_VAC.fb_SP1K1_MONO_VGC_2.i_xOpnLS
//     PlcTask Outputs/GVL_SXR_VAC.fb_SP1K1_MONO_VGC_2.q_xOPN_DO <-> Channel 11/GVL_SXR_VAC.fb_SP1K1_MONO_VGC_2.q_xOPN_DO
//   SxrVacPlc/SxrVacPlc Instance <-> =+-EK1200_00_00-CPU/EtherCAT1/=+-EP2338_09_03
//     PlcTask Inputs/GVL_SXR_VAC.fb_IM1K2_PPM_VGC_1.i_xClsLS <-> Channel 2/GVL_SXR_VAC.fb_IM1K2_PPM_VGC_1.i_xClsLS
//     PlcTask Inputs/GVL_SXR_VAC.fb_IM1K2_PPM_VGC_1.i_xOpnLS <-> Channel 1/GVL_SXR_VAC.fb_IM1K2_PPM_VGC_1.i_xOpnLS
//     PlcTask Inputs/GVL_SXR_VAC.fb_TV3K0_VGC_1.i_xClsLS <-> Channel 6/GVL_SXR_VAC.fb_TV3K0_VGC_1.i_xClsLS
//     PlcTask Inputs/GVL_SXR_VAC.fb_TV3K0_VGC_1.i_xOpnLS <-> Channel 5/GVL_SXR_VAC.fb_TV3K0_VGC_1.i_xOpnLS
//     PlcTask Outputs/GVL_SXR_VAC.fb_IM1K2_PPM_VGC_1.q_xOPN_DO <-> Channel 11/GVL_SXR_VAC.fb_IM1K2_PPM_VGC_1.q_xOPN_DO
//     PlcTask Outputs/GVL_SXR_VAC.fb_TV3K0_VGC_1.q_xOPN_DO <-> Channel 15/GVL_SXR_VAC.fb_TV3K0_VGC_1.q_xOPN_DO
//   SxrVacPlc/SxrVacPlc Instance <-> =+-EK1200_00_00-CPU/EtherCAT1/=+-EP2338_10_02
//     PlcTask Inputs/GVL_SXR_VAC.fb_MR1K4_SOMS_VGC_1.i_xClsLS <-> Channel 2/GVL_SXR_VAC.fb_MR1K4_SOMS_VGC_1.i_xClsLS
//     PlcTask Inputs/GVL_SXR_VAC.fb_MR1K4_SOMS_VGC_1.i_xOpnLS <-> Channel 1/GVL_SXR_VAC.fb_MR1K4_SOMS_VGC_1.i_xOpnLS
//     PlcTask Outputs/GVL_SXR_VAC.fb_MR1K4_SOMS_VGC_1.q_xOPN_DO <-> Channel 11/GVL_SXR_VAC.fb_MR1K4_SOMS_VGC_1.q_xOPN_DO
//   SxrVacPlc/SxrVacPlc Instance <-> =+-EK1200_00_00-CPU/EtherCAT1/=+-EP2338_11_02
//     PlcTask Inputs/GVL_SXR_VAC.fb_TV1K4_VGC_1.i_xClsLS <-> Channel 2/GVL_SXR_VAC.fb_TV1K4_VGC_1.i_xClsLS
//     PlcTask Inputs/GVL_SXR_VAC.fb_TV1K4_VGC_2.i_xClsLS <-> Channel 6/GVL_SXR_VAC.fb_TV1K4_VGC_2.i_xClsLS
//     PlcTask Inputs/GVL_SXR_VAC.fb_TV1K4_VGC_1.i_xOpnLS <-> Channel 1/GVL_SXR_VAC.fb_TV1K4_VGC_1.i_xOpnLS
//     PlcTask Inputs/GVL_SXR_VAC.fb_TV1K4_VGC_2.i_xOpnLS <-> Channel 5/GVL_SXR_VAC.fb_TV1K4_VGC_2.i_xOpnLS
//     PlcTask Outputs/GVL_SXR_VAC.fb_TV1K4_VGC_1.q_xOPN_DO <-> Channel 11/GVL_SXR_VAC.fb_TV1K4_VGC_1.q_xOPN_DO
//     PlcTask Outputs/GVL_SXR_VAC.fb_TV1K4_VGC_2.q_xOPN_DO <-> Channel 15/GVL_SXR_VAC.fb_TV1K4_VGC_2.q_xOPN_DO
//   SxrVacPlc/SxrVacPlc Instance <-> =+-EK1200_00_00-CPU/EtherCAT1/=+-EP2338_14_00
//     PlcTask Inputs/GVL_SXR_VAC.fb_ST3K4_XTES_VGC_1.i_xClsLS <-> Channel 2/GVL_SXR_VAC.fb_ST3K4_XTES_VGC_1.i_xClsLS
//     PlcTask Inputs/GVL_SXR_VAC.fb_ST3K4_XTES_VGC_1.i_xOpnLS <-> Channel 1/GVL_SXR_VAC.fb_ST3K4_XTES_VGC_1.i_xOpnLS
//     PlcTask Outputs/GVL_SXR_VAC.fb_ST3K4_XTES_VGC_1.q_xOPN_DO <-> Channel 11/GVL_SXR_VAC.fb_ST3K4_XTES_VGC_1.q_xOPN_DO
//   SxrVacPlc/SxrVacPlc Instance <-> =+-EK1200_00_00-CPU/EtherCAT1/=+-EP2624_07_02
//     PlcTask Outputs/GVL_SXR_VAC.fb_MR1K3_TXI_GCC_1.q_xHV_DIS <-> Channel 1/GVL_SXR_VAC.fb_MR1K3_TXI_GCC_1.q_xHV_DIS
//   SxrVacPlc/SxrVacPlc Instance <-> =+-EK1200_00_00-CPU/EtherCAT1/=+-EP2624_08_02
//     PlcTask Outputs/GVL_SXR_VAC.fb_MR2K3_TXI_GCC_1.q_xHV_DIS <-> Channel 1/GVL_SXR_VAC.fb_MR2K3_TXI_GCC_1.q_xHV_DIS
//   SxrVacPlc/SxrVacPlc Instance <-> =+-EK1200_00_00-CPU/EtherCAT1/=+-EP2624_09_01
//     PlcTask Outputs/GVL_SXR_VAC.fb_SP1K1_MONO_GCC_1.q_xHV_DIS <-> Channel 1/GVL_SXR_VAC.fb_SP1K1_MONO_GCC_1.q_xHV_DIS
//   SxrVacPlc/SxrVacPlc Instance <-> =+-EK1200_00_00-CPU/EtherCAT1/=+-EP2624_10_01
//     PlcTask Outputs/GVL_SXR_VAC.fb_TV3K0_GCC_1.q_xHV_DIS <-> Channel 1/GVL_SXR_VAC.fb_TV3K0_GCC_1.q_xHV_DIS
//   SxrVacPlc/SxrVacPlc Instance <-> =+-EK1200_00_00-CPU/EtherCAT1/=+-EP2624_11_01
//     PlcTask Outputs/GVL_SXR_VAC.fb_MR1K4_SOMS_GCC_1.q_xHV_DIS <-> Channel 2/GVL_SXR_VAC.fb_MR1K4_SOMS_GCC_1.q_xHV_DIS
//     PlcTask Outputs/GVL_SXR_VAC.fb_TV1K4_GCC_1.q_xHV_DIS <-> Channel 1/GVL_SXR_VAC.fb_TV1K4_GCC_1.q_xHV_DIS
//   SxrVacPlc/SxrVacPlc Instance <-> =+-EK1200_00_00-CPU/EtherCAT1/=+-EP2624_12_01
//     PlcTask Outputs/GVL_SXR_VAC.fb_ST1K4_TEST_GCC_1.q_xHV_DIS <-> Channel 1/GVL_SXR_VAC.fb_ST1K4_TEST_GCC_1.q_xHV_DIS
//   SxrVacPlc/SxrVacPlc Instance <-> =+-EK1200_00_00-CPU/EtherCAT1/=+-EP2624_13_01
//     PlcTask Outputs/GVL_SXR_VAC.fb_ST2K4_BCS_GCC_1.q_xHV_DIS <-> Channel 1/GVL_SXR_VAC.fb_ST2K4_BCS_GCC_1.q_xHV_DIS
//   SxrVacPlc/SxrVacPlc Instance <-> =+-EK1200_00_00-CPU/EtherCAT1/=+-EP2624_14_02
//     PlcTask Outputs/GVL_SXR_VAC.fb_PC4K4_XTES_GCC_1.q_xHV_DIS <-> Channel 1/GVL_SXR_VAC.fb_PC4K4_XTES_GCC_1.q_xHV_DIS
//   SxrVacPlc/SxrVacPlc Instance <-> =+-EK1200_00_00-CPU/EtherCAT1/=+-EP3174_07_01
//     PlcTask Inputs/GVL_SXR_VAC.fb_MR1K3_TXI_GCC_1.i_iPRESS_R <-> AI Standard Channel 2/GVL_SXR_VAC.fb_MR1K3_TXI_GCC_1.i_iPRESS_R
//     PlcTask Inputs/GVL_SXR_VAC.fb_MR1K3_TXI_GPI_1.i_iPRESS_R <-> AI Standard Channel 1/GVL_SXR_VAC.fb_MR1K3_TXI_GPI_1.i_iPRESS_R
//   SxrVacPlc/SxrVacPlc Instance <-> =+-EK1200_00_00-CPU/EtherCAT1/=+-EP3174_08_01
//     PlcTask Inputs/GVL_SXR_VAC.fb_MR2K3_TXI_GCC_1.i_iPRESS_R <-> AI Standard Channel 2/GVL_SXR_VAC.fb_MR2K3_TXI_GCC_1.i_iPRESS_R
//     PlcTask Inputs/GVL_SXR_VAC.fb_MR2K3_TXI_GPI_1.i_iPRESS_R <-> AI Standard Channel 1/GVL_SXR_VAC.fb_MR2K3_TXI_GPI_1.i_iPRESS_R
//   SxrVacPlc/SxrVacPlc Instance <-> =+-EK1200_00_00-CPU/EtherCAT1/=+-EP3174_09_00
//     PlcTask Inputs/GVL_SXR_VAC.fb_SP1K1_MONO_GCC_1.i_iPRESS_R <-> AI Standard Channel 1/GVL_SXR_VAC.fb_SP1K1_MONO_GCC_1.i_iPRESS_R
//     PlcTask Inputs/GVL_SXR_VAC.fb_SP1K1_MONO_GPI_1.i_iPRESS_R <-> AI Standard Channel 2/GVL_SXR_VAC.fb_SP1K1_MONO_GPI_1.i_iPRESS_R
//   SxrVacPlc/SxrVacPlc Instance <-> =+-EK1200_00_00-CPU/EtherCAT1/=+-EP3174_10_00
//     PlcTask Inputs/GVL_SXR_VAC.fb_MR1K4_SOMS_GPI_1.i_iPRESS_R <-> AI Standard Channel 2/GVL_SXR_VAC.fb_MR1K4_SOMS_GPI_1.i_iPRESS_R
//     PlcTask Inputs/GVL_SXR_VAC.fb_TV3K0_GCC_1.i_iPRESS_R <-> AI Standard Channel 1/GVL_SXR_VAC.fb_TV3K0_GCC_1.i_iPRESS_R
//     PlcTask Inputs/GVL_SXR_VAC.fb_TV3K0_GPI_1.i_iPRESS_R <-> AI Standard Channel 4/GVL_SXR_VAC.fb_TV3K0_GPI_1.i_iPRESS_R
//   SxrVacPlc/SxrVacPlc Instance <-> =+-EK1200_00_00-CPU/EtherCAT1/=+-EP3174_11_00
//     PlcTask Inputs/GVL_SXR_VAC.fb_MR1K4_SOMS_GCC_1.i_iPRESS_R <-> AI Standard Channel 3/GVL_SXR_VAC.fb_MR1K4_SOMS_GCC_1.i_iPRESS_R
//     PlcTask Inputs/GVL_SXR_VAC.fb_TV1K4_GCC_1.i_iPRESS_R <-> AI Standard Channel 2/GVL_SXR_VAC.fb_TV1K4_GCC_1.i_iPRESS_R
//     PlcTask Inputs/GVL_SXR_VAC.fb_TV1K4_GPI_1.i_iPRESS_R <-> AI Standard Channel 1/GVL_SXR_VAC.fb_TV1K4_GPI_1.i_iPRESS_R
//   SxrVacPlc/SxrVacPlc Instance <-> =+-EK1200_00_00-CPU/EtherCAT1/=+-EP3174_12_00
//     PlcTask Inputs/GVL_SXR_VAC.fb_ST1K4_TEST_GCC_1.i_iPRESS_R <-> AI Standard Channel 2/GVL_SXR_VAC.fb_ST1K4_TEST_GCC_1.i_iPRESS_R
//     PlcTask Inputs/GVL_SXR_VAC.fb_ST1K4_TEST_GPI_1.i_iPRESS_R <-> AI Standard Channel 1/GVL_SXR_VAC.fb_ST1K4_TEST_GPI_1.i_iPRESS_R
//   SxrVacPlc/SxrVacPlc Instance <-> =+-EK1200_00_00-CPU/EtherCAT1/=+-EP3174_13_00
//     PlcTask Inputs/GVL_SXR_VAC.fb_ST2K4_BCS_GCC_1.i_iPRESS_R <-> AI Standard Channel 2/GVL_SXR_VAC.fb_ST2K4_BCS_GCC_1.i_iPRESS_R
//     PlcTask Inputs/GVL_SXR_VAC.fb_ST2K4_BCS_GPI_1.i_iPRESS_R <-> AI Standard Channel 1/GVL_SXR_VAC.fb_ST2K4_BCS_GPI_1.i_iPRESS_R
//   SxrVacPlc/SxrVacPlc Instance <-> =+-EK1200_00_00-CPU/EtherCAT1/=+-EP3174_14_01
//     PlcTask Inputs/GVL_SXR_VAC.fb_PC4K4_XTES_GCC_1.i_iPRESS_R <-> AI Standard Channel 2/GVL_SXR_VAC.fb_PC4K4_XTES_GCC_1.i_iPRESS_R
//     PlcTask Inputs/GVL_SXR_VAC.fb_PC4K4_XTES_GPI_1.i_iPRESS_R <-> AI Standard Channel 1/GVL_SXR_VAC.fb_PC4K4_XTES_GPI_1.i_iPRESS_R
//   SxrVacSim/SxrVacSim Instance <-> SimDevice 2 (EtherCAT Simulation)/=+-EL2798_01_02
//     SimTask Inputs/GVL_SXR_VAC.st_DMPS_GCC_1.i_xHvOn <-> Channel 1/GVL_SXR_VAC.fb_DMPS_GCC_1.q_xHV_DIS
//     SimTask Inputs/GVL_SXR_VAC.st_IM2K0_XTES_GCC_1.i_xHvOn <-> Channel 2/GVL_SXR_VAC.fb_IM2K0_XTES_GCC_1.q_xHV_DIS
//     SimTask Inputs/GVL_SXR_VAC.st_PCPM3B_GFS_1.i_xHvOn <-> Channel 5/GVL_SXR_VAC.fb_PCPM3B_GFS_1.q_xHV_DIS
//     SimTask Inputs/GVL_SXR_VAC.st_SL1K0_GCC_1.i_xHvOn <-> Channel 4/GVL_SXR_VAC.fb_SL1K0_GCC_1.q_xHV_DIS
//   SxrVacSim/SxrVacSim Instance <-> SimDevice 2 (EtherCAT Simulation)/=+-EL2798_01_06
//     SimTask Inputs/GVL_SXR_VAC.st_MR1K1_BEND_GCC_1.i_xHvOn <-> Channel 5/GVL_SXR_VAC.fb_MR1K1_BEND_GCC_1.q_xHV_DIS
//     SimTask Inputs/GVL_SXR_VAC.st_PA1K0_GCC_1.i_xHvOn <-> Channel 4/GVL_SXR_VAC.fb_PA1K0_GCC_1.q_xHV_DIS
//     SimTask Inputs/GVL_SXR_VAC.st_TV2K0_GCC_1.i_xHvOn <-> Channel 1/GVL_SXR_VAC.fb_TV2K0_GCC_1.q_xHV_DIS
//     SimTask Inputs/GVL_SXR_VAC.st_TV2K0_GCC_2.i_xHvOn <-> Channel 2/GVL_SXR_VAC.fb_TV2K0_GCC_2.q_xHV_DIS
//   SxrVacSim/SxrVacSim Instance <-> SimDevice 2 (EtherCAT Simulation)/=+-ES3068_01_01
//     SimTask Outputs/GVL_SXR_VAC.st_DMPS_GCC_1.q_iRawPress <-> AI Standard Channel 1/GVL_SXR_VAC.fb_DMPS_GCC_1.i_iPRESS_R
//     SimTask Outputs/GVL_SXR_VAC.st_DMPS_GPI_1.q_iRawPress <-> AI Standard Channel 5/GVL_SXR_VAC.fb_DMPS_GPI_1.i_iPRESS_R
//     SimTask Outputs/GVL_SXR_VAC.st_IM2K0_XTES_GCC_1.q_iRawPress <-> AI Standard Channel 3/GVL_SXR_VAC.fb_IM2K0_XTES_GCC_1.i_iPRESS_R
//     SimTask Outputs/GVL_SXR_VAC.st_IM2K0_XTES_GPI_1.q_iRawPress <-> AI Standard Channel 6/GVL_SXR_VAC.fb_IM2K0_XTES_GPI_1.i_iPRESS_R
//   SxrVacSim/SxrVacSim Instance <-> SimDevice 2 (EtherCAT Simulation)/=+-ES3068_01_04
//     SimTask Outputs/GVL_SXR_VAC.st_PCPM3B_GFS_1.q_iRawPress <-> AI Standard Channel 3/GVL_SXR_VAC.fb_PCPM3B_GFS_1.i_iPRESS_R
//     SimTask Outputs/GVL_SXR_VAC.st_SL1K0_GCC_1.q_iRawPress <-> AI Standard Channel 1/GVL_SXR_VAC.fb_SL1K0_GCC_1.i_iPRESS_R
//     SimTask Outputs/GVL_SXR_VAC.st_SL1K0_GPI_1.q_iRawPress <-> AI Standard Channel 5/GVL_SXR_VAC.fb_SL1K0_GPI_1.i_iPRESS_R
//   SxrVacSim/SxrVacSim Instance <-> SimDevice 2 (EtherCAT Simulation)/=+-ES3068_01_05
//     SimTask Outputs/GVL_SXR_VAC.st_TV2K0_GCC_1.q_iRawPress <-> AI Standard Channel 1/GVL_SXR_VAC.fb_TV2K0_GCC_1.i_iPRESS_R
//     SimTask Outputs/GVL_SXR_VAC.st_TV2K0_GCC_2.q_iRawPress <-> AI Standard Channel 3/GVL_SXR_VAC.fb_TV2K0_GCC_2.i_iPRESS_R
//     SimTask Outputs/GVL_SXR_VAC.st_TV2K0_GPI_1.q_iRawPress <-> AI Standard Channel 5/GVL_SXR_VAC.fb_TV2K0_GPI_1.i_iPRESS_R
//     SimTask Outputs/GVL_SXR_VAC.st_TV2K0_GPI_2.q_iRawPress <-> AI Standard Channel 6/GVL_SXR_VAC.fb_TV2K0_GPI_2.i_iPRESS_R
//   SxrVacSim/SxrVacSim Instance <-> SimDevice 2 (EtherCAT Simulation)/=+-ES3068_01_08
//     SimTask Outputs/GVL_SXR_VAC.st_MR1K1_BEND_GCC_1.q_iRawPress <-> AI Standard Channel 3/GVL_SXR_VAC.fb_MR1K1_BEND_GCC_1.i_iPRESS_R
//     SimTask Outputs/GVL_SXR_VAC.st_MR1K1_BEND_GPI_1.q_iRawPress <-> AI Standard Channel 6/GVL_SXR_VAC.fb_MR1K1_BEND_GPI_1.i_iPRESS_R
//     SimTask Outputs/GVL_SXR_VAC.st_PA1K0_GCC_1.q_iRawPress <-> AI Standard Channel 1/GVL_SXR_VAC.fb_PA1K0_GCC_1.i_iPRESS_R
//     SimTask Outputs/GVL_SXR_VAC.st_PA1K0_GPI_1.q_iRawPress <-> AI Standard Channel 5/GVL_SXR_VAC.fb_PA1K0_GPI_1.i_iPRESS_R
//   SxrVacSim/SxrVacSim Instance <-> SimDevice 2 (EtherCAT Simulation)/=+-ES1004_03_01
//     SimTask Outputs/GVL_SXR_VAC.st_EM1K0_GMD_VGC_1.q_xClsLS <-> Channel 4/GVL_SXR_VAC.fb_EM1K0_GMD_VGC_1.i_xClsLS
//     SimTask Outputs/GVL_SXR_VAC.st_EM1K0_GMD_VGC_1.q_xOpnLS <-> Channel 3/GVL_SXR_VAC.fb_EM1K0_GMD_VGC_1.i_xOpnLS
//     SimTask Outputs/GVL_SXR_VAC.st_RTDSK0_VGC_1.q_xClsLS <-> Channel 2/GVL_SXR_VAC.fb_RTDSK0_VGC_1.i_xClsLS
//     SimTask Outputs/GVL_SXR_VAC.st_RTDSK0_VGC_1.q_xOpnLS <-> Channel 1/GVL_SXR_VAC.fb_RTDSK0_VGC_1.i_xOpnLS
//   SxrVacSim/SxrVacSim Instance <-> SimDevice 2 (EtherCAT Simulation)/=+-ES1004_03_04
//     SimTask Outputs/GVL_SXR_VAC.st_AT1K0_GAS_VGC_1.q_xClsLS <-> Channel 2/GVL_SXR_VAC.fb_AT1K0_GAS_VGC_1.i_xClsLS
//     SimTask Outputs/GVL_SXR_VAC.st_AT1K0_GAS_VGC_1.q_xOpnLS <-> Channel 1/GVL_SXR_VAC.fb_AT1K0_GAS_VGC_1.i_xOpnLS
//   SxrVacSim/SxrVacSim Instance <-> SimDevice 2 (EtherCAT Simulation)/=+-ES2004_03_02
//     SimTask Inputs/GVL_SXR_VAC.st_EM1K0_GMD_VGC_1.i_xSol <-> Channel 3/GVL_SXR_VAC.fb_EM1K0_GMD_VGC_1.q_xOPN_DO
//     SimTask Inputs/GVL_SXR_VAC.st_RTDSK0_VGC_1.i_xSol <-> Channel 1/GVL_SXR_VAC.fb_RTDSK0_VGC_1.q_xOPN_DO
//   SxrVacSim/SxrVacSim Instance <-> SimDevice 2 (EtherCAT Simulation)/=+-ES2004_03_03
//     SimTask Inputs/GVL_SXR_VAC.st_AT1K0_GAS_VGC_1.i_xSol <-> Channel 1/GVL_SXR_VAC.fb_AT1K0_GAS_VGC_1.q_xOPN_DO
//   SxrVacSim/SxrVacSim Instance <-> SimDevice 2 (EtherCAT Simulation)/=+-EL2794_15_03
//     SimTask Inputs/GVL_SXR_VAC.st_MR1K4_SOMS_PIP_1.xOn <-> Channel 1/GVL_SXR_VAC.fb_MR1K4_SOMS_PIP_1.q_xHVEna_DO
//     SimTask Inputs/GVL_SXR_VAC.st_ST1K4_TEST_PIP_1.xOn <-> Channel 2/GVL_SXR_VAC.fb_ST1K4_TEST_PIP_1.q_xHVEna_DO
//     SimTask Inputs/GVL_SXR_VAC.st_ST2K4_BCS_PIP_1.xOn <-> Channel 3/GVL_SXR_VAC.fb_ST2K4_BCS_PIP_1.q_xHVEna_DO
//     SimTask Inputs/GVL_SXR_VAC.st_ST3K4_PPS_PIP_1.xOn <-> Channel 4/GVL_SXR_VAC.fb_ST3K4_PPS_PIP_1.q_xHVEna_DO
//   SxrVacSim/SxrVacSim Instance <-> SimDevice 2 (EtherCAT Simulation)/=+-EL2794_15_06
//     SimTask Inputs/GVL_SXR_VAC.st_PC4K4_XTES_PIP_1.xOn <-> Channel 1/GVL_SXR_VAC.fb_PC4K4_XTES_PIP_1.q_xHVEna_DO
//   SxrVacSim/SxrVacSim Instance <-> SimDevice 2 (EtherCAT Simulation)/=+-EL2794_00_03
//     SimTask Inputs/GVL_SXR_VAC.st_RTDSK0_PIP_{1..4}.xOn <-> Channel {1..4}/GVL_SXR_VAC.fb_RTDSK0_PIP_{1..4}.q_xHVEna_DO  (4 links)
//   SxrVacSim/SxrVacSim Instance <-> SimDevice 2 (EtherCAT Simulation)/=+-EL2794_00_06
//     SimTask Inputs/GVL_SXR_VAC.st_PCPM3B_PIP_1.xOn <-> Channel 2/GVL_SXR_VAC.fb_PCPM3B_PIP_1.q_xHVEna_DO
//     SimTask Inputs/GVL_SXR_VAC.st_RTDSK0_PIP_5.xOn <-> Channel 1/GVL_SXR_VAC.fb_RTDSK0_PIP_5.q_xHVEna_DO
//   SxrVacSim/SxrVacSim Instance <-> SimDevice 2 (EtherCAT Simulation)/=+-EL2794_00_10
//     SimTask Inputs/GVL_SXR_VAC.st_MR1K1_BEND_PIP_1.xOn <-> Channel 3/GVL_SXR_VAC.fb_MR1K1_BEND_PIP_1.q_xHVEna_DO
//     SimTask Inputs/GVL_SXR_VAC.st_MR1K3_TXI_PIP_1.xOn <-> Channel 4/GVL_SXR_VAC.fb_MR1K3_TXI_PIP_1.q_xHVEna_DO
//     SimTask Inputs/GVL_SXR_VAC.st_PA1K0_PIP_1.xOn <-> Channel 1/GVL_SXR_VAC.fb_PA1K0_PIP_1.q_xHVEna_DO
//   SxrVacSim/SxrVacSim Instance <-> SimDevice 2 (EtherCAT Simulation)/=+-EL2794_00_13
//     SimTask Inputs/GVL_SXR_VAC.st_MR2K3_TXI_PIP_1.xOn <-> Channel 1/GVL_SXR_VAC.fb_MR2K3_TXI_PIP_1.q_xHVEna_DO
//     SimTask Inputs/GVL_SXR_VAC.st_SP1K1_MONO_PIP_1.xOn <-> Channel 2/GVL_SXR_VAC.fb_SP1K1_MONO_PIP_1.q_xHVEna_DO
//     SimTask Inputs/GVL_SXR_VAC.st_SP1K1_MONO_PIP_2.xOn <-> Channel 3/GVL_SXR_VAC.fb_SP1K1_MONO_PIP_2.q_xHVEna_DO
//     SimTask Inputs/GVL_SXR_VAC.st_TV3K0_PIP_1.xOn <-> Channel 4/GVL_SXR_VAC.fb_TV3K0_PIP_1.q_xHVEna_DO
//   SxrVacSim/SxrVacSim Instance <-> SimDevice 2 (EtherCAT Simulation)/=+-EP2338_04_00
//     SimTask Outputs/GVL_SXR_VAC.st_EM1K0_XGMD_VGC_1.q_xClsLS <-> Channel 2/GVL_SXR_VAC.fb_EM1K0_XGMD_VGC_1.i_xClsLS
//     SimTask Outputs/GVL_SXR_VAC.st_EM1K0_XGMD_VGC_2.q_xClsLS <-> Channel 6/GVL_SXR_VAC.fb_EM1K0_XGMD_VGC_2.i_xClsLS
//     SimTask Outputs/GVL_SXR_VAC.st_EM1K0_XGMD_VGC_1.q_xOpnLS <-> Channel 1/GVL_SXR_VAC.fb_EM1K0_XGMD_VGC_1.i_xOpnLS
//     SimTask Outputs/GVL_SXR_VAC.st_EM1K0_XGMD_VGC_2.q_xOpnLS <-> Channel 5/GVL_SXR_VAC.fb_EM1K0_XGMD_VGC_2.i_xOpnLS
//     SimTask Inputs/GVL_SXR_VAC.st_EM1K0_XGMD_VGC_1.i_xSol <-> Channel 11/GVL_SXR_VAC.fb_EM1K0_XGMD_VGC_1.q_xOPN_DO
//     SimTask Inputs/GVL_SXR_VAC.st_EM1K0_XGMD_VGC_2.i_xSol <-> Channel 15/GVL_SXR_VAC.fb_EM1K0_XGMD_VGC_2.q_xOPN_DO
//   SxrVacSim/SxrVacSim Instance <-> SimDevice 2 (EtherCAT Simulation)/=+-EP2338_05_00
//     SimTask Outputs/GVL_SXR_VAC.st_TV2K0_VGC_1.q_xClsLS <-> Channel 2/GVL_SXR_VAC.fb_TV2K0_VGC_1.i_xClsLS
//     SimTask Outputs/GVL_SXR_VAC.st_TV2K0_VGC_1.q_xOpnLS <-> Channel 1/GVL_SXR_VAC.fb_TV2K0_VGC_1.i_xOpnLS
//     SimTask Inputs/GVL_SXR_VAC.st_TV2K0_VGC_1.i_xSol <-> Channel 11/GVL_SXR_VAC.fb_TV2K0_VGC_1.q_xOPN_DO
//   SxrVacSim/SxrVacSim Instance <-> SimDevice 2 (EtherCAT Simulation)/=+-EP2338_06_00
//     SimTask Outputs/GVL_SXR_VAC.st_MR1K1_BEND_VGC_1.q_xClsLS <-> Channel 2/GVL_SXR_VAC.fb_MR1K1_BEND_VGC_1.i_xClsLS
//     SimTask Outputs/GVL_SXR_VAC.st_MR1K1_BEND_VGC_1.q_xOpnLS <-> Channel 1/GVL_SXR_VAC.fb_MR1K1_BEND_VGC_1.i_xOpnLS
//     SimTask Inputs/GVL_SXR_VAC.st_MR1K1_BEND_VGC_1.i_xSol <-> Channel 11/GVL_SXR_VAC.fb_MR1K1_BEND_VGC_1.q_xOPN_DO
//   SxrVacSim/SxrVacSim Instance <-> SimDevice 2 (EtherCAT Simulation)/=+-EP2338_07_00
//     SimTask Outputs/GVL_SXR_VAC.st_MR1K3_TXI_VGC_1.q_xClsLS <-> Channel 2/GVL_SXR_VAC.fb_MR1K3_TXI_VGC_1.i_xClsLS
//     SimTask Outputs/GVL_SXR_VAC.st_MR1K3_TXI_VGC_1.q_xOpnLS <-> Channel 1/GVL_SXR_VAC.fb_MR1K3_TXI_VGC_1.i_xOpnLS
//     SimTask Inputs/GVL_SXR_VAC.st_MR1K3_TXI_VGC_1.i_xSol <-> Channel 11/GVL_SXR_VAC.fb_MR1K3_TXI_VGC_1.q_xOPN_DO
//   SxrVacSim/SxrVacSim Instance <-> SimDevice 2 (EtherCAT Simulation)/=+-EP2338_08_00
//     SimTask Outputs/GVL_SXR_VAC.st_SP1K1_MONO_VGC_1.q_xClsLS <-> Channel 2/GVL_SXR_VAC.fb_SP1K1_MONO_VGC_1.i_xClsLS
//     SimTask Outputs/GVL_SXR_VAC.st_SP1K1_MONO_VGC_1.q_xOpnLS <-> Channel 1/GVL_SXR_VAC.fb_SP1K1_MONO_VGC_1.i_xOpnLS
//     SimTask Inputs/GVL_SXR_VAC.st_SP1K1_MONO_VGC_1.i_xSol <-> Channel 11/GVL_SXR_VAC.fb_SP1K1_MONO_VGC_1.q_xOPN_DO
//   SxrVacSim/SxrVacSim Instance <-> SimDevice 2 (EtherCAT Simulation)/=+-EP2338_09_02
//     SimTask Outputs/GVL_SXR_VAC.st_SP1K1_MONO_VGC_2.q_xClsLS <-> Channel 2/GVL_SXR_VAC.fb_SP1K1_MONO_VGC_2.i_xClsLS
//     SimTask Outputs/GVL_SXR_VAC.st_SP1K1_MONO_VGC_2.q_xOpnLS <-> Channel 1/GVL_SXR_VAC.fb_SP1K1_MONO_VGC_2.i_xOpnLS
//     SimTask Inputs/GVL_SXR_VAC.st_SP1K1_MONO_VGC_2.i_xSol <-> Channel 11/GVL_SXR_VAC.fb_SP1K1_MONO_VGC_2.q_xOPN_DO
//   SxrVacSim/SxrVacSim Instance <-> SimDevice 2 (EtherCAT Simulation)/=+-EP2338_09_03
//     SimTask Outputs/GVL_SXR_VAC.st_IM1K2_PPM_VGC_1.q_xClsLS <-> Channel 2/GVL_SXR_VAC.fb_IM1K2_PPM_VGC_1.i_xClsLS
//     SimTask Outputs/GVL_SXR_VAC.st_IM1K2_PPM_VGC_1.q_xOpnLS <-> Channel 1/GVL_SXR_VAC.fb_IM1K2_PPM_VGC_1.i_xOpnLS
//     SimTask Outputs/GVL_SXR_VAC.st_TV3K0_VGC_1.q_xClsLS <-> Channel 6/GVL_SXR_VAC.fb_TV3K0_VGC_1.i_xClsLS
//     SimTask Outputs/GVL_SXR_VAC.st_TV3K0_VGC_1.q_xOpnLS <-> Channel 5/GVL_SXR_VAC.fb_TV3K0_VGC_1.i_xOpnLS
//     SimTask Inputs/GVL_SXR_VAC.st_IM1K2_PPM_VGC_1.i_xSol <-> Channel 11/GVL_SXR_VAC.fb_IM1K2_PPM_VGC_1.q_xOPN_DO
//     SimTask Inputs/GVL_SXR_VAC.st_TV3K0_VGC_1.i_xSol <-> Channel 15/GVL_SXR_VAC.fb_TV3K0_VGC_1.q_xOPN_DO
//   SxrVacSim/SxrVacSim Instance <-> SimDevice 2 (EtherCAT Simulation)/=+-EP2338_10_02
//     SimTask Outputs/GVL_SXR_VAC.st_MR1K4_SOMS_VGC_1.q_xClsLS <-> Channel 2/GVL_SXR_VAC.fb_MR1K4_SOMS_VGC_1.i_xClsLS
//     SimTask Outputs/GVL_SXR_VAC.st_MR1K4_SOMS_VGC_1.q_xOpnLS <-> Channel 1/GVL_SXR_VAC.fb_MR1K4_SOMS_VGC_1.i_xOpnLS
//     SimTask Inputs/GVL_SXR_VAC.st_MR1K4_SOMS_VGC_1.i_xSol <-> Channel 11/GVL_SXR_VAC.fb_MR1K4_SOMS_VGC_1.q_xOPN_DO
//   SxrVacSim/SxrVacSim Instance <-> SimDevice 2 (EtherCAT Simulation)/=+-EP2338_11_02
//     SimTask Outputs/GVL_SXR_VAC.st_TV1K4_VGC_1.q_xClsLS <-> Channel 2/GVL_SXR_VAC.fb_TV1K4_VGC_1.i_xClsLS
//     SimTask Outputs/GVL_SXR_VAC.st_TV1K4_VGC_2.q_xClsLS <-> Channel 6/GVL_SXR_VAC.fb_TV1K4_VGC_2.i_xClsLS
//     SimTask Outputs/GVL_SXR_VAC.st_TV1K4_VGC_1.q_xOpnLS <-> Channel 1/GVL_SXR_VAC.fb_TV1K4_VGC_1.i_xOpnLS
//     SimTask Outputs/GVL_SXR_VAC.st_TV1K4_VGC_2.q_xOpnLS <-> Channel 5/GVL_SXR_VAC.fb_TV1K4_VGC_2.i_xOpnLS
//     SimTask Inputs/GVL_SXR_VAC.st_TV1K4_VGC_1.i_xSol <-> Channel 11/GVL_SXR_VAC.fb_TV1K4_VGC_1.q_xOPN_DO
//     SimTask Inputs/GVL_SXR_VAC.st_TV1K4_VGC_2.i_xSol <-> Channel 15/GVL_SXR_VAC.fb_TV1K4_VGC_2.q_xOPN_DO
//   SxrVacSim/SxrVacSim Instance <-> SimDevice 2 (EtherCAT Simulation)/=+-EP2338_14_00
//     SimTask Outputs/GVL_SXR_VAC.st_ST3K4_XTES_VGC_1.q_xClsLS <-> Channel 2/GVL_SXR_VAC.fb_ST3K4_XTES_VGC_1.i_xClsLS
//     SimTask Outputs/GVL_SXR_VAC.st_ST3K4_XTES_VGC_1.q_xOpnLS <-> Channel 1/GVL_SXR_VAC.fb_ST3K4_XTES_VGC_1.i_xOpnLS
//     SimTask Inputs/GVL_SXR_VAC.st_ST3K4_XTES_VGC_1.i_xSol <-> Channel 11/GVL_SXR_VAC.fb_ST3K4_XTES_VGC_1.q_xOPN_DO
//   SxrVacSim/SxrVacSim Instance <-> SimDevice 2 (EtherCAT Simulation)/=+-EP2624_07_02
//     SimTask Inputs/GVL_SXR_VAC.st_MR1K3_TXI_GCC_1.i_xHvOn <-> Channel 1/GVL_SXR_VAC.fb_MR1K3_TXI_GCC_1.q_xHV_DIS
//   SxrVacSim/SxrVacSim Instance <-> SimDevice 2 (EtherCAT Simulation)/=+-EP2624_08_02
//     SimTask Inputs/GVL_SXR_VAC.st_MR2K3_TXI_GCC_1.i_xHvOn <-> Channel 1/GVL_SXR_VAC.fb_MR2K3_TXI_GCC_1.q_xHV_DIS
//   SxrVacSim/SxrVacSim Instance <-> SimDevice 2 (EtherCAT Simulation)/=+-EP2624_09_01
//     SimTask Inputs/GVL_SXR_VAC.st_SP1K1_MONO_GCC_1.i_xHvOn <-> Channel 1/GVL_SXR_VAC.fb_SP1K1_MONO_GCC_1.q_xHV_DIS
//   SxrVacSim/SxrVacSim Instance <-> SimDevice 2 (EtherCAT Simulation)/=+-EP2624_10_01
//     SimTask Inputs/GVL_SXR_VAC.st_TV3K0_GCC_1.i_xHvOn <-> Channel 1/GVL_SXR_VAC.fb_TV3K0_GCC_1.q_xHV_DIS
//   SxrVacSim/SxrVacSim Instance <-> SimDevice 2 (EtherCAT Simulation)/=+-EP2624_11_01
//     SimTask Inputs/GVL_SXR_VAC.st_MR1K4_SOMS_GCC_1.i_xHvOn <-> Channel 2/GVL_SXR_VAC.fb_MR1K4_SOMS_GCC_1.q_xHV_DIS
//     SimTask Inputs/GVL_SXR_VAC.st_TV1K4_GCC_1.i_xHvOn <-> Channel 1/GVL_SXR_VAC.fb_TV1K4_GCC_1.q_xHV_DIS
//   SxrVacSim/SxrVacSim Instance <-> SimDevice 2 (EtherCAT Simulation)/=+-EP2624_12_01
//     SimTask Inputs/GVL_SXR_VAC.st_ST1K4_TEST_GCC_1.i_xHvOn <-> Channel 1/GVL_SXR_VAC.fb_ST1K4_TEST_GCC_1.q_xHV_DIS
//   SxrVacSim/SxrVacSim Instance <-> SimDevice 2 (EtherCAT Simulation)/=+-EP2624_13_01
//     SimTask Inputs/GVL_SXR_VAC.st_ST2K4_BCS_GCC_1.i_xHvOn <-> Channel 1/GVL_SXR_VAC.fb_ST2K4_BCS_GCC_1.q_xHV_DIS
//   SxrVacSim/SxrVacSim Instance <-> SimDevice 2 (EtherCAT Simulation)/=+-EP2624_14_02
//     SimTask Inputs/GVL_SXR_VAC.st_PC4K4_XTES_GCC_1.i_xHvOn <-> Channel 1/GVL_SXR_VAC.fb_PC4K4_XTES_GCC_1.q_xHV_DIS
//   SxrVacSim/SxrVacSim Instance <-> SimDevice 2 (EtherCAT Simulation)/=+-EP3174_07_01
//     SimTask Outputs/GVL_SXR_VAC.st_MR1K3_TXI_GCC_1.q_iRawPress <-> AI Standard Channel 2/GVL_SXR_VAC.fb_MR1K3_TXI_GCC_1.i_iPRESS_R
//     SimTask Outputs/GVL_SXR_VAC.st_MR1K3_TXI_GPI_1.q_iRawPress <-> AI Standard Channel 1/GVL_SXR_VAC.fb_MR1K3_TXI_GPI_1.i_iPRESS_R
//   SxrVacSim/SxrVacSim Instance <-> SimDevice 2 (EtherCAT Simulation)/=+-EP3174_08_01
//     SimTask Outputs/GVL_SXR_VAC.st_MR2K3_TXI_GCC_1.q_iRawPress <-> AI Standard Channel 2/GVL_SXR_VAC.fb_MR2K3_TXI_GCC_1.i_iPRESS_R
//     SimTask Outputs/GVL_SXR_VAC.st_MR2K3_TXI_GPI_1.q_iRawPress <-> AI Standard Channel 1/GVL_SXR_VAC.fb_MR2K3_TXI_GPI_1.i_iPRESS_R
//   SxrVacSim/SxrVacSim Instance <-> SimDevice 2 (EtherCAT Simulation)/=+-EP3174_09_00
//     SimTask Outputs/GVL_SXR_VAC.st_SP1K1_MONO_GCC_1.q_iRawPress <-> AI Standard Channel 1/GVL_SXR_VAC.fb_SP1K1_MONO_GCC_1.i_iPRESS_R
//     SimTask Outputs/GVL_SXR_VAC.st_SP1K1_MONO_GPI_1.q_iRawPress <-> AI Standard Channel 2/GVL_SXR_VAC.fb_SP1K1_MONO_GPI_1.i_iPRESS_R
//   SxrVacSim/SxrVacSim Instance <-> SimDevice 2 (EtherCAT Simulation)/=+-EP3174_10_00
//     SimTask Outputs/GVL_SXR_VAC.st_MR1K4_SOMS_GPI_1.q_iRawPress <-> AI Standard Channel 2/GVL_SXR_VAC.fb_MR1K4_SOMS_GPI_1.i_iPRESS_R
//     SimTask Outputs/GVL_SXR_VAC.st_TV3K0_GCC_1.q_iRawPress <-> AI Standard Channel 1/GVL_SXR_VAC.fb_TV3K0_GCC_1.i_iPRESS_R
//     SimTask Outputs/GVL_SXR_VAC.st_TV3K0_GPI_1.q_iRawPress <-> AI Standard Channel 4/GVL_SXR_VAC.fb_TV3K0_GPI_1.i_iPRESS_R
//   SxrVacSim/SxrVacSim Instance <-> SimDevice 2 (EtherCAT Simulation)/=+-EP3174_11_00
//     SimTask Outputs/GVL_SXR_VAC.st_MR1K4_SOMS_GCC_1.q_iRawPress <-> AI Standard Channel 3/GVL_SXR_VAC.fb_MR1K4_SOMS_GCC_1.i_iPRESS_R
//     SimTask Outputs/GVL_SXR_VAC.st_TV1K4_GCC_1.q_iRawPress <-> AI Standard Channel 2/GVL_SXR_VAC.fb_TV1K4_GCC_1.i_iPRESS_R
//     SimTask Outputs/GVL_SXR_VAC.st_TV1K4_GPI_1.q_iRawPress <-> AI Standard Channel 1/GVL_SXR_VAC.fb_TV1K4_GPI_1.i_iPRESS_R
//   SxrVacSim/SxrVacSim Instance <-> SimDevice 2 (EtherCAT Simulation)/=+-EP3174_12_00
//     SimTask Outputs/GVL_SXR_VAC.st_ST1K4_TEST_GCC_1.q_iRawPress <-> AI Standard Channel 2/GVL_SXR_VAC.fb_ST1K4_TEST_GCC_1.i_iPRESS_R
//     SimTask Outputs/GVL_SXR_VAC.st_ST1K4_TEST_GPI_1.q_iRawPress <-> AI Standard Channel 1/GVL_SXR_VAC.fb_ST1K4_TEST_GPI_1.i_iPRESS_R
//   SxrVacSim/SxrVacSim Instance <-> SimDevice 2 (EtherCAT Simulation)/=+-EP3174_13_00
//     SimTask Outputs/GVL_SXR_VAC.st_ST2K4_BCS_GCC_1.q_iRawPress <-> AI Standard Channel 2/GVL_SXR_VAC.fb_ST2K4_BCS_GCC_1.i_iPRESS_R
//     SimTask Outputs/GVL_SXR_VAC.st_ST2K4_BCS_GPI_1.q_iRawPress <-> AI Standard Channel 1/GVL_SXR_VAC.fb_ST2K4_BCS_GPI_1.i_iPRESS_R
//   SxrVacSim/SxrVacSim Instance <-> SimDevice 2 (EtherCAT Simulation)/=+-EP3174_14_01
//     SimTask Outputs/GVL_SXR_VAC.st_PC4K4_XTES_GCC_1.q_iRawPress <-> AI Standard Channel 2/GVL_SXR_VAC.fb_PC4K4_XTES_GCC_1.i_iPRESS_R
//     SimTask Outputs/GVL_SXR_VAC.st_PC4K4_XTES_GPI_1.q_iRawPress <-> AI Standard Channel 1/GVL_SXR_VAC.fb_PC4K4_XTES_GPI_1.i_iPRESS_R

CONFIGURATION SxrVacPlc
    RESOURCE PLC ON TwinCAT3
        TASK PlcTask(INTERVAL := T#10ms, PRIORITY := 20);
        PROGRAM MAIN WITH PlcTask : MAIN;
    END_RESOURCE
END_CONFIGURATION

// ---- GVLs/GVL_SXR_VAC.TcGVL
VAR_GLOBAL


// MKS275 Gauges

{attribute 'pytmc' := ' pv: MR2K3:TXI:GPI:1 '}
fb_MR2K3_TXI_GPI_1 : FB_MKS275;
{attribute 'pytmc' := ' pv: MR1K3:TXI:GPI:1 '}
fb_MR1K3_TXI_GPI_1 : FB_MKS275;
{attribute 'pytmc' := ' pv: SP1K1:MONO:GPI:1 '}
fb_SP1K1_MONO_GPI_1 : FB_MKS275;
{attribute 'pytmc' := ' pv: TV3K0:GPI:1 '}
fb_TV3K0_GPI_1 : FB_MKS275;
{attribute 'pytmc' := ' pv: MR1K4:SOMS:GPI:1 '}
fb_MR1K4_SOMS_GPI_1 : FB_MKS275;
{attribute 'pytmc' := ' pv: TV1K4:GPI:1 '}
fb_TV1K4_GPI_1 : FB_MKS275;
{attribute 'pytmc' := ' pv: ST1K4:TEST:GPI:1 '}
fb_ST1K4_TEST_GPI_1 : FB_MKS275;
{attribute 'pytmc' := ' pv: ST2K4:BCS:GPI:1 '}
fb_ST2K4_BCS_GPI_1 : FB_MKS275;
{attribute 'pytmc' := ' pv: PC4K4:XTES:GPI:1 '}
fb_PC4K4_XTES_GPI_1 : FB_MKS275;

// MKS500_EP Gauges

{attribute 'pytmc' := ' pv: MR2K3:TXI:GCC:1 '}
fb_MR2K3_TXI_GCC_1 : FB_MKS500_EP;
{attribute 'pytmc' := ' pv: MR1K3:TXI:GCC:1 '}
fb_MR1K3_TXI_GCC_1 : FB_MKS500_EP;
{attribute 'pytmc' := ' pv: SP1K1:MONO:GCC:1 '}
fb_SP1K1_MONO_GCC_1 : FB_MKS500_EP;
{attribute 'pytmc' := ' pv: TV3K0:GCC:1 '}
fb_TV3K0_GCC_1 : FB_MKS500_EP;
{attribute 'pytmc' := ' pv: MR1K4:SOMS:GCC:1 '}
fb_MR1K4_SOMS_GCC_1 : FB_MKS500_EP;
{attribute 'pytmc' := ' pv: TV1K4:GCC:1 '}
fb_TV1K4_GCC_1 : FB_MKS500_EP;
{attribute 'pytmc' := ' pv: ST1K4:TEST:GCC:1 '}
fb_ST1K4_TEST_GCC_1 : FB_MKS500_EP;
{attribute 'pytmc' := ' pv: ST2K4:BCS:GCC:1 '}
fb_ST2K4_BCS_GCC_1 : FB_MKS500_EP;
{attribute 'pytmc' := ' pv: PC4K4:XTES:GCC:1 '}
fb_PC4K4_XTES_GCC_1 : FB_MKS500_EP;

// VGC Valves

{attribute 'pytmc' := ' pv: RTDSK0:VGC:1 '}
fb_RTDSK0_VGC_1 : FB_VGC;
{attribute 'pytmc' := ' pv: EM1K0:GMD:VGC:1 '}
fb_EM1K0_GMD_VGC_1 : FB_VGC;
{attribute 'pytmc' := ' pv: AT1K0:GAS:VGC:1 '}
fb_AT1K0_GAS_VGC_1 : FB_VGC;
{attribute 'pytmc' := ' pv: EM1K0:XGMD:VGC:1 '}
fb_EM1K0_XGMD_VGC_1 : FB_VGC;
{attribute 'pytmc' := ' pv: EM1K0:XGMD:VGC:2 '}
fb_EM1K0_XGMD_VGC_2 : FB_VGC;
{attribute 'pytmc' := ' pv: TV2K0:VGC:1 '}
fb_TV2K0_VGC_1 : FB_VGC;
{attribute 'pytmc' := ' pv: MR1K1:BEND:VGC:1 '}
fb_MR1K1_BEND_VGC_1 : FB_VGC;
{attribute 'pytmc' := ' pv: MR1K3:TXI:VGC:1 '}
fb_MR1K3_TXI_VGC_1 : FB_VGC;
{attribute 'pytmc' := ' pv: SP1K1:MONO:VGC:1 '}
fb_SP1K1_MONO_VGC_1 : FB_VGC;
{attribute 'pytmc' := ' pv: SP1K1:MONO:VGC:2 '}
fb_SP1K1_MONO_VGC_2 : FB_VGC;
{attribute 'pytmc' := ' pv: IM1K2:PPM:VGC:1 '}
fb_IM1K2_PPM_VGC_1 : FB_VGC;
{attribute 'pytmc' := ' pv: TV3K0:VGC:1 '}
fb_TV3K0_VGC_1 : FB_VGC;
{attribute 'pytmc' := ' pv: MR1K4:SOMS:VGC:1 '}
fb_MR1K4_SOMS_VGC_1 : FB_VGC;
{attribute 'pytmc' := ' pv: TV1K4:VGC:1 '}
fb_TV1K4_VGC_1 : FB_VGC;
{attribute 'pytmc' := ' pv: TV1K4:VGC:2 '}
fb_TV1K4_VGC_2 : FB_VGC;
{attribute 'pytmc' := ' pv: ST3K4:XTES:VGC:1 '}
fb_ST3K4_XTES_VGC_1 : FB_VGC;

// PIP_Gamma Pumps

{attribute 'pytmc' := ' pv: RTDSK0:PIP:1 '}
fb_RTDSK0_PIP_1 : FB_PIP_GAMMA;
{attribute 'pytmc' := ' pv: RTDSK0:PIP:2 '}
fb_RTDSK0_PIP_2 : FB_PIP_GAMMA;
{attribute 'pytmc' := ' pv: RTDSK0:PIP:3 '}
fb_RTDSK0_PIP_3 : FB_PIP_GAMMA;
{attribute 'pytmc' := ' pv: RTDSK0:PIP:4 '}
fb_RTDSK0_PIP_4 : FB_PIP_GAMMA;
{attribute 'pytmc' := ' pv: RTDSK0:PIP:5 '}
fb_RTDSK0_PIP_5 : FB_PIP_GAMMA;
{attribute 'pytmc' := ' pv: PCPM3B:PIP:1 '}
fb_PCPM3B_PIP_1 : FB_PIP_GAMMA;
{attribute 'pytmc' := ' pv: PA1K0:PIP:1 '}
fb_PA1K0_PIP_1 : FB_PIP_GAMMA;
{attribute 'pytmc' := ' pv: PA1K0 '}
fb_PA1K0 : FB_PIP_GAMMA;
{attribute 'pytmc' := ' pv: MR1K1:BEND:PIP:1 '}
fb_MR1K1_BEND_PIP_1 : FB_PIP_GAMMA;
{attribute 'pytmc' := ' pv: MR2K3:TXI:PIP:1 '}
fb_MR2K3_TXI_PIP_1 : FB_PIP_GAMMA;
{attribute 'pytmc' := ' pv: MR1K3:TXI:PIP:1 '}
fb_MR1K3_TXI_PIP_1 : FB_PIP_GAMMA;
{attribute 'pytmc' := ' pv: SP1K1:MONO:PIP:1 '}
fb_SP1K1_MONO_PIP_1 : FB_PIP_GAMMA;
{attribute 'pytmc' := ' pv: SP1K1:MONO:PIP:2 '}
fb_SP1K1_MONO_PIP_2 : FB_PIP_GAMMA;
{attribute 'pytmc' := ' pv: TV3K0:PIP:1 '}
fb_TV3K0_PIP_1 : FB_PIP_GAMMA;
{attribute 'pytmc' := ' pv: MR1K4:SOMS:PIP:1 '}
fb_MR1K4_SOMS_PIP_1 : FB_PIP_GAMMA;
{attribute 'pytmc' := ' pv: ST1K4:TEST:PIP:1 '}
fb_ST1K4_TEST_PIP_1 : FB_PIP_GAMMA;
{attribute 'pytmc' := ' pv: ST2K4:BCS:PIP:1 '}
fb_ST2K4_BCS_PIP_1 : FB_PIP_GAMMA;
{attribute 'pytmc' := ' pv: ST3K4:PPS:PIP:1 '}
fb_ST3K4_PPS_PIP_1 : FB_PIP_GAMMA;
{attribute 'pytmc' := ' pv: PC4K4:XTES:PIP:1 '}
fb_PC4K4_XTES_PIP_1 : FB_PIP_GAMMA;

// FB_MKS422

{attribute 'pytmc' := ' pv: DMPS:GCC:1 '}
fb_DMPS_GCC_1 : FB_MKS422;
{attribute 'pytmc' := ' pv: IM2K0:XTES:GCC:1 '}
fb_IM2K0_XTES_GCC_1 : FB_MKS422;
{attribute 'pytmc' := ' pv: PCPM3B:GFS:1 '}
fb_PCPM3B_GFS_1 : FB_MKS422;
{attribute 'pytmc' := ' pv: SL1K0:GCC:1 '}
fb_SL1K0_GCC_1 : FB_MKS422;
{attribute 'pytmc' := ' pv: TV2K0:GCC:1 '}
fb_TV2K0_GCC_1 : FB_MKS422;
{attribute 'pytmc' := ' pv: TV2K0:GCC:2 '}
fb_TV2K0_GCC_2 : FB_MKS422;
{attribute 'pytmc' := ' pv: PA1K0:GCC:1 '}
fb_PA1K0_GCC_1 : FB_MKS422;
{attribute 'pytmc' := ' pv: MR1K1:BEND:GCC:1 '}
fb_MR1K1_BEND_GCC_1 : FB_MKS422;

// FB_MKS317

{attribute 'pytmc' := ' pv: DMPS:GPI:1 '}
fb_DMPS_GPI_1 : FB_MKS317;
{attribute 'pytmc' := ' pv: IM2K0:XTES:GPI:1 '}
fb_IM2K0_XTES_GPI_1 : FB_MKS317;
{attribute 'pytmc' := ' pv: SL1K0:GPI:1 '}
fb_SL1K0_GPI_1 : FB_MKS317;
{attribute 'pytmc' := ' pv: TV2K0:GPI:1 '}
fb_TV2K0_GPI_1 : FB_MKS317;
{attribute 'pytmc' := ' pv: TV2K0:GPI:2 '}
fb_TV2K0_GPI_2 : FB_MKS317;
{attribute 'pytmc' := ' pv: PA1K0:GPI:1 '}
fb_PA1K0_GPI_1 : FB_MKS317;
{attribute 'pytmc' := ' pv: MR1K1:BEND:GPI:1 '}
fb_MR1K1_BEND_GPI_1 : FB_MKS317;

END_VAR

// ---- GVLs/GVL_Variables.TcGVL
VAR_GLOBAL

xSystemOverrideMode : BOOL; (* Global system override for the prototype section*)

END_VAR

// ---- POUs/MAIN.TcPOU
PROGRAM MAIN
VAR
END_VAR

PRG_DIAGNOSTIC();
PRG_SXR_VAC();

END_PROGRAM

// ---- POUs/PRG_DIAGNOSTIC.TcPOU
PROGRAM PRG_DIAGNOSTIC
VAR

   fbTime : FB_LocalSystemTime := ( bEnable := TRUE, dwCycle := 1 );
   logTimer : TON := ( IN := TRUE, PT := T#1000ms );

   plcName : STRING[15];

   {attribute 'pytmc' := ' pv: simHeartbeat '}
   simHeartbeat AT %I* : UINT := 0;
   {attribute 'pytmc' := ' pv: plcHeartbeat '}
   plcHeartbeat : UDINT := 0;
   {attribute 'pytmc' := ' pv: plcInfo '}
   plcInfo : STRING[40];
   {attribute 'pytmc' := ' pv: plcLocalTime '}
   plcLocalTime : STRING[25];

END_VAR

plcHeartbeat := plcHeartbeat + 1;
IF plcHeartbeat > 4294967000
   THEN plcHeartbeat := 0;
END_IF

// get timestamp as string every second
fbTime();
logTimer( IN := fbTime.bValid );
IF logTimer.Q THEN
   logTimer( IN := FALSE ); logTimer( IN := fbTime.bValid );
   plcLocalTime := SYSTEMTIME_TO_STRING(fbTime.systemTime);
END_IF

// make an info string
plcName := 'Prototype PLC: ';
plcInfo := CONCAT(plcName, plcLocalTime);

END_PROGRAM

// ---- POUs/PRG_SXR_VAC.TcPOU
PROGRAM PRG_SXR_VAC
VAR
END_VAR


// MKS275 Gauges

fb_MR2K3_TXI_GPI_1(PG=>);
fb_MR1K3_TXI_GPI_1(PG=>);
fb_SP1K1_MONO_GPI_1(PG=>);
fb_TV3K0_GPI_1(PG=>);
fb_MR1K4_SOMS_GPI_1(PG=>);
fb_TV1K4_GPI_1(PG=>);
fb_ST1K4_TEST_GPI_1(PG=>);
fb_ST2K4_BCS_GPI_1(PG=>);
fb_PC4K4_XTES_GPI_1(PG=>);

// MKS500_EP Gauges

fb_MR2K3_TXI_GCC_1(PG := fb_MR2K3_TXI_GPI_1.PG);
fb_MR1K3_TXI_GCC_1(PG := fb_MR1K3_TXI_GPI_1.PG);
fb_SP1K1_MONO_GCC_1(PG := fb_SP1K1_MONO_GPI_1.PG);
fb_TV3K0_GCC_1(PG := fb_TV3K0_GPI_1.PG);
fb_MR1K4_SOMS_GCC_1(PG := fb_MR1K4_SOMS_GPI_1.PG);
fb_TV1K4_GCC_1(PG := fb_TV1K4_GPI_1.PG);
fb_ST1K4_TEST_GCC_1(PG := fb_ST1K4_TEST_GPI_1.PG);
fb_ST2K4_BCS_GCC_1(PG := fb_ST2K4_BCS_GPI_1.PG);
fb_PC4K4_XTES_GCC_1(PG := fb_PC4K4_XTES_GPI_1.PG);

// VGC Valves

fb_RTDSK0_VGC_1(i_stUSG := fb_DMPS_GCC_1.IG, i_stDSG := , i_xDis_DPIlk := FALSE, i_xEPS_OK := TRUE, i_xPMPS_OK := TRUE, i_xExt_OK := TRUE, i_xOverrideMode := xSystemOverrideMode);
fb_EM1K0_GMD_VGC_1(i_stUSG := fb_DMPS_GCC_1.IG, i_stDSG := , i_xDis_DPIlk := FALSE, i_xEPS_OK := TRUE, i_xPMPS_OK := TRUE, i_xExt_OK := TRUE, i_xOverrideMode := xSystemOverrideMode);
fb_AT1K0_GAS_VGC_1(i_stUSG := , i_stDSG := , i_xDis_DPIlk := FALSE, i_xEPS_OK := TRUE, i_xPMPS_OK := TRUE, i_xExt_OK := TRUE, i_xOverrideMode := xSystemOverrideMode);
fb_EM1K0_XGMD_VGC_1(i_stUSG := , i_stDSG := , i_xDis_DPIlk := FALSE, i_xEPS_OK := TRUE, i_xPMPS_OK := TRUE, i_xExt_OK := TRUE, i_xOverrideMode := xSystemOverrideMode);
fb_EM1K0_XGMD_VGC_2(i_stUSG := , i_stDSG := fb_TV2K0_GCC_1.IG, i_xDis_DPIlk := FALSE, i_xEPS_OK := TRUE, i_xPMPS_OK := TRUE, i_xExt_OK := TRUE, i_xOverrideMode := xSystemOverrideMode);
fb_TV2K0_VGC_1(i_stUSG := fb_TV2K0_GCC_1.IG, i_stDSG := fb_TV2K0_GCC_2.IG, i_xDis_DPIlk := FALSE, i_xEPS_OK := TRUE, i_xPMPS_OK := TRUE, i_xExt_OK := TRUE, i_xOverrideMode := xSystemOverrideMode);
fb_MR1K1_BEND_VGC_1(i_stUSG := fb_PA1K0_GCC_1.IG, i_stDSG := fb_MR1K1_BEND_GCC_1.IG, i_xDis_DPIlk := FALSE, i_xEPS_OK := TRUE, i_xPMPS_OK := TRUE, i_xExt_OK := TRUE, i_xOverrideMode := xSystemOverrideMode);
fb_MR1K3_TXI_VGC_1(i_stUSG := fb_MR1K1_BEND_GCC_1.IG, i_stDSG := fb_MR1K3_TXI_GCC_1.IG, i_xDis_DPIlk := FALSE, i_xEPS_OK := TRUE, i_xPMPS_OK := TRUE, i_xExt_OK := TRUE, i_xOverrideMode := xSystemOverrideMode);
fb_SP1K1_MONO_VGC_1(i_stUSG := fb_MR2K3_TXI_GCC_1.IG, i_stDSG := fb_SP1K1_MONO_GCC_1.IG, i_xDis_DPIlk := FALSE, i_xEPS_OK := TRUE, i_xPMPS_OK := TRUE, i_xExt_OK := TRUE, i_xOverrideMode := xSystemOverrideMode);
fb_SP1K1_MONO_VGC_2(i_stUSG := fb_MR2K3_TXI_GCC_1.IG, i_stDSG := , i_xDis_DPIlk := FALSE, i_xEPS_OK := TRUE, i_xPMPS_OK := TRUE, i_xExt_OK := TRUE, i_xOverrideMode := xSystemOverrideMode);
fb_IM1K2_PPM_VGC_1(i_stUSG := fb_MR2K3_TXI_GCC_1.IG, i_stDSG := , i_xDis_DPIlk := FALSE, i_xEPS_OK := TRUE, i_xPMPS_OK := TRUE, i_xExt_OK := TRUE, i_xOverrideMode := xSystemOverrideMode);
fb_TV3K0_VGC_1(i_stUSG := fb_MR2K3_TXI_GCC_1.IG, i_stDSG := fb_TV3K0_GCC_1.IG, i_xDis_DPIlk := FALSE, i_xEPS_OK := TRUE, i_xPMPS_OK := TRUE, i_xExt_OK := TRUE, i_xOverrideMode := xSystemOverrideMode);
fb_MR1K4_SOMS_VGC_1(i_stUSG := fb_TV3K0_GCC_1.IG, i_stDSG := fb_MR1K4_SOMS_GCC_1.IG, i_xDis_DPIlk := FALSE, i_xEPS_OK := TRUE, i_xPMPS_OK := TRUE, i_xExt_OK := TRUE, i_xOverrideMode := xSystemOverrideMode);
fb_TV1K4_VGC_1(i_stUSG := fb_MR1K4_SOMS_GCC_1.IG, i_stDSG := fb_TV1K4_GCC_1.IG, i_xDis_DPIlk := FALSE, i_xEPS_OK := TRUE, i_xPMPS_OK := TRUE, i_xExt_OK := TRUE, i_xOverrideMode := xSystemOverrideMode);
fb_TV1K4_VGC_2(i_stUSG := fb_TV1K4_GCC_1.IG, i_stDSG := fb_ST1K4_TEST_GCC_1.IG, i_xDis_DPIlk := FALSE, i_xEPS_OK := TRUE, i_xPMPS_OK := TRUE, i_xExt_OK := TRUE, i_xOverrideMode := xSystemOverrideMode);
fb_ST3K4_XTES_VGC_1(i_stUSG := fb_ST2K4_BCS_GCC_1.IG, i_stDSG := fb_PC4K4_XTES_GCC_1.IG, i_xDis_DPIlk := FALSE, i_xEPS_OK := TRUE, i_xPMPS_OK := TRUE, i_xExt_OK := TRUE, i_xOverrideMode := xSystemOverrideMode);

// PIP_Gamma Pumps

fb_RTDSK0_PIP_1(i_stGauge := fb_DMPS_GCC_1.PG);
fb_RTDSK0_PIP_2(i_stGauge := fb_DMPS_GCC_1.PG);
fb_RTDSK0_PIP_3(i_stGauge := fb_DMPS_GCC_1.PG);
fb_RTDSK0_PIP_4(i_stGauge := fb_DMPS_GCC_1.PG);
fb_RTDSK0_PIP_5(i_stGauge := fb_DMPS_GCC_1.PG);
fb_PCPM3B_PIP_1(i_stGauge := fb_IM2K0_XTES_GCC_1.PG);
fb_PA1K0_PIP_1(i_stGauge := fb_PA1K0_GCC_1.PG);
fb_PA1K0(i_stGauge := fb_PA1K0_GCC_1.PG);
fb_MR1K1_BEND_PIP_1(i_stGauge := fb_MR1K1_BEND_GCC_1.PG);
fb_MR2K3_TXI_PIP_1(i_stGauge := fb_MR2K3_TXI_GCC_1.PG);
fb_MR1K3_TXI_PIP_1(i_stGauge := fb_MR1K3_TXI_GCC_1.PG);
fb_SP1K1_MONO_PIP_1(i_stGauge := fb_SP1K1_MONO_GCC_1.PG);
fb_SP1K1_MONO_PIP_2(i_stGauge := fb_SP1K1_MONO_GCC_1.PG);
fb_TV3K0_PIP_1(i_stGauge := fb_TV3K0_GCC_1.PG);
fb_MR1K4_SOMS_PIP_1(i_stGauge := fb_MR1K4_SOMS_GCC_1.PG);
fb_ST1K4_TEST_PIP_1(i_stGauge := fb_ST1K4_TEST_GCC_1.PG);
fb_ST2K4_BCS_PIP_1(i_stGauge := fb_ST2K4_BCS_GCC_1.PG);
fb_ST3K4_PPS_PIP_1(i_stGauge := fb_ST2K4_BCS_GCC_1.PG);
fb_PC4K4_XTES_PIP_1(i_stGauge := fb_PC4K4_XTES_GCC_1.PG);

// FB_MKS422

fb_DMPS_GCC_1(PG := fb_DMPS_GPI_1.PG);
fb_IM2K0_XTES_GCC_1(PG := fb_IM2K0_XTES_GPI_1.PG);
fb_PCPM3B_GFS_1(PG := fb_SL1K0_GPI_1.PG);
fb_SL1K0_GCC_1(PG := fb_SL1K0_GPI_1.PG);
fb_TV2K0_GCC_1(PG := fb_TV2K0_GPI_1.PG);
fb_TV2K0_GCC_2(PG := fb_TV2K0_GPI_1.PG);
fb_PA1K0_GCC_1(PG := fb_PA1K0_GPI_1.PG);
fb_MR1K1_BEND_GCC_1(PG := fb_MR1K1_BEND_GPI_1.PG);

// FB_MKS317

fb_DMPS_GPI_1(PG=>);
fb_IM2K0_XTES_GPI_1(PG=>);
fb_SL1K0_GPI_1(PG=>);
fb_TV2K0_GPI_1(PG=>);
fb_TV2K0_GPI_2(PG=>);
fb_PA1K0_GPI_1(PG=>);
fb_MR1K1_BEND_GPI_1(PG=>);

END_PROGRAM
